LIN {X 0.053,Y -179.837,Z 893.459,A 0.000,B 0.000,C 90.000,E1 262.648} C_DIS
LIN {X -0.069,Y -179.024,Z 893.445,A 0.000,B 0.000,C 90.000,E1 260.151} C_DIS
LIN {X -0.006,Y -178.664,Z 893.440,A 0.000,B 0.000,C 90.000,E1 259.285} C_DIS
LIN {X -0.070,Y -175.715,Z 893.412,A 0.000,B 0.000,C 90.000,E1 254.212} C_DIS
LIN {X -0.053,Y -172.430,Z 893.388,A 0.000,B 0.000,C 90.000,E1 249.934} C_DIS
LIN {X -0.035,Y -171.257,Z 893.379,A 0.000,B 0.000,C 90.000,E1 248.209} C_DIS
LIN {X -0.051,Y -167.530,Z 893.355,A 0.000,B 0.000,C 90.000,E1 243.896} C_DIS
LIN {X 0.033,Y -166.925,Z 893.350,A 0.000,B 0.000,C 90.000,E1 242.999} C_DIS
LIN {X -0.046,Y -162.921,Z 893.326,A 0.000,B 0.000,C 90.000,E1 238.663} C_DIS
LIN {X -0.068,Y -161.594,Z 893.316,A 0.000,B 0.000,C 90.000,E1 236.914} C_DIS
LIN {X 0.057,Y -158.336,Z 893.296,A 0.000,B 0.000,C 90.000,E1 233.336} C_DIS
LIN {X -0.081,Y -155.638,Z 893.277,A 0.000,B 0.000,C 90.000,E1 229.828} C_DIS
LIN {X -0.027,Y -151.912,Z 893.252,A 0.000,B 0.000,C 90.000,E1 225.324} C_DIS
LIN {X -0.012,Y -150.145,Z 893.237,A 0.000,B 0.000,C 90.000,E1 222.609} C_DIS
LIN {X 0.025,Y -146.929,Z 893.211,A 0.000,B 0.000,C 90.000,E1 218.051} C_DIS
LIN {X 0.017,Y -145.517,Z 893.196,A 0.000,B 0.000,C 90.000,E1 215.311} C_DIS
LIN {X 0.011,Y -142.917,Z 893.171,A 0.000,B 0.000,C 90.000,E1 210.718} C_DIS
LIN {X 0.064,Y -141.540,Z 893.150,A 0.000,B 0.000,C 90.000,E1 207.001} C_DIS
LIN {X -0.024,Y -139.402,Z 893.114,A 0.000,B 0.000,C 90.000,E1 200.536} C_DIS
LIN {X -0.019,Y -139.118,Z 893.104,A 0.000,B 0.000,C 90.000,E1 198.671} C_DIS
LIN {X 0.012,Y -138.352,Z 893.057,A 0.000,B 0.000,C 90.000,E1 190.254} C_DIS
LIN {X 0.002,Y -139.505,Z 893.005,A 0.000,B 0.000,C 90.000,E1 180.917} C_DIS
LIN {X -0.057,Y -141.138,Z 892.974,A 0.000,B 0.000,C 90.000,E1 175.355} C_DIS
LIN {X 0.037,Y -142.518,Z 892.959,A 0.000,B 0.000,C 90.000,E1 172.534} C_DIS
LIN {X -0.018,Y -144.781,Z 892.933,A 0.000,B 0.000,C 90.000,E1 167.937} C_DIS
LIN {X -0.029,Y -147.396,Z 892.913,A 0.000,B 0.000,C 90.000,E1 164.267} C_DIS
LIN {X 0.001,Y -149.971,Z 892.892,A 0.000,B 0.000,C 90.000,E1 160.604} C_DIS
LIN {X 0.012,Y -153.292,Z 892.872,A 0.000,B 0.000,C 90.000,E1 156.975} C_DIS
LIN {X -0.001,Y -154.996,Z 892.862,A 0.000,B 0.000,C 90.000,E1 155.177} C_DIS
LIN {X 0.012,Y -158.636,Z 892.842,A 0.000,B 0.000,C 90.000,E1 151.591} C_DIS
LIN {X -0.051,Y -161.910,Z 892.827,A 0.000,B 0.000,C 90.000,E1 148.948} C_DIS
LIN {X 0.056,Y -166.101,Z 892.808,A 0.000,B 0.000,C 90.000,E1 145.388} C_DIS
LIN {X 0.054,Y -171.110,Z 892.788,A 0.000,B 0.000,C 90.000,E1 141.904} C_DIS
LIN {X -0.026,Y -175.985,Z 892.769,A 0.000,B 0.000,C 90.000,E1 138.485} C_DIS
LIN {X 0.088,Y -180.231,Z 892.755,A 0.000,B 0.000,C 90.000,E1 135.891} C_DIS
LIN {X 0.061,Y -185.646,Z 892.736,A 0.000,B 0.000,C 90.000,E1 132.528} C_DIS
LIN {X 0.115,Y -190.245,Z 892.722,A 0.000,B 0.000,C 90.000,E1 130.011} C_DIS
LIN {X -0.048,Y -193.381,Z 892.712,A 0.000,B 0.000,C 90.000,E1 128.222} C_DIS
LIN {X 0.109,Y -294.897,Z 892.712,A 0.000,B 0.000,C 90.000,E1 128.177} C_DIS
LIN {X 0.093,Y -299.925,Z 892.711,A 0.000,B 0.000,C 90.000,E1 128.016} C_DIS
LIN {X -0.060,Y -302.135,Z 892.710,A 0.000,B 0.000,C 90.000,E1 127.890} C_DIS
LIN {X 0.005,Y -305.159,Z 892.709,A 0.000,B 0.000,C 90.000,E1 127.569} C_DIS
LIN {X -0.008,Y -308.784,Z 892.706,A 0.000,B 0.000,C 90.000,E1 126.996} C_DIS
LIN {X 0.017,Y -310.226,Z 892.704,A 0.000,B 0.000,C 90.000,E1 126.664} C_DIS
LIN {X -0.023,Y -311.357,Z 892.702,A 0.000,B 0.000,C 90.000,E1 126.343} C_DIS
LIN {X 0.139,Y -321.511,Z 892.684,A 0.000,B 0.000,C 90.000,E1 123.086} C_DIS
LIN {X 0.013,Y -331.967,Z 892.668,A 0.000,B 0.000,C 90.000,E1 120.256} C_DIS
LIN {X -0.023,Y -343.778,Z 892.653,A 0.000,B 0.000,C 90.000,E1 117.462} C_DIS
LIN {X -0.023,Y -357.045,Z 892.637,A 0.000,B 0.000,C 90.000,E1 114.719} C_DIS
LIN {X -0.034,Y -370.158,Z 892.624,A 0.000,B 0.000,C 90.000,E1 112.333} C_DIS
LIN {X -0.006,Y -384.610,Z 892.611,A 0.000,B 0.000,C 90.000,E1 109.993} C_DIS
LIN {X 0.121,Y -400.503,Z 892.598,A 0.000,B 0.000,C 90.000,E1 107.692} C_DIS
LIN {X 0.017,Y -417.952,Z 892.586,A 0.000,B 0.000,C 90.000,E1 105.481} C_DIS
LIN {X 0.148,Y -437.059,Z 892.574,A 0.000,B 0.000,C 90.000,E1 103.300} C_DIS
LIN {X -0.056,Y -457.177,Z 892.563,A 0.000,B 0.000,C 90.000,E1 101.299} C_DIS
LIN {X -0.201,Y -467.395,Z 892.557,A 0.000,B 0.000,C 90.000,E1 100.366} C_DIS
LIN {X -0.258,Y -469.394,Z 892.556,A 0.000,B 0.000,C 90.000,E1 100.141} C_DIS
LIN {X 0.054,Y -471.044,Z 892.555,A 0.000,B 0.000,C 90.000,E1 99.849} C_DIS
LIN {X -0.099,Y -472.281,Z 892.553,A 0.000,B 0.000,C 90.000,E1 99.613} C_DIS
LIN {X 0.005,Y -473.801,Z 892.551,A 0.000,B 0.000,C 90.000,E1 99.095} C_DIS
LIN {X 0.191,Y -474.280,Z 892.548,A 0.000,B 0.000,C 90.000,E1 98.568} C_DIS
LIN {X -0.155,Y -473.796,Z 892.545,A 0.000,B 0.000,C 90.000,E1 98.106} C_DIS
LIN {X -0.028,Y -472.278,Z 892.542,A 0.000,B 0.000,C 90.000,E1 97.587} C_DIS
LIN {X -0.169,Y -471.051,Z 892.541,A 0.000,B 0.000,C 90.000,E1 97.352} C_DIS
LIN {X 0.203,Y -452.056,Z 892.524,A 0.000,B 0.000,C 90.000,E1 94.245} C_DIS
LIN {X 0.123,Y -443.002,Z 892.515,A 0.000,B 0.000,C 90.000,E1 92.694} C_DIS
LIN {X -0.134,Y -433.515,Z 892.506,A 0.000,B 0.000,C 90.000,E1 91.146} C_DIS
LIN {X -0.125,Y -423.861,Z 892.497,A 0.000,B 0.000,C 90.000,E1 89.542} C_DIS
LIN {X -0.091,Y -410.897,Z 892.485,A 0.000,B 0.000,C 90.000,E1 87.364} C_DIS
LIN {X 0.014,Y -399.646,Z 892.475,A 0.000,B 0.000,C 90.000,E1 85.412} C_DIS
LIN {X -0.043,Y -386.908,Z 892.462,A 0.000,B 0.000,C 90.000,E1 83.166} C_DIS
LIN {X 0.063,Y -375.774,Z 892.451,A 0.000,B 0.000,C 90.000,E1 81.141} C_DIS
LIN {X -0.003,Y -364.602,Z 892.439,A 0.000,B 0.000,C 90.000,E1 79.106} C_DIS
LIN {X -0.188,Y -354.940,Z 892.430,A 0.000,B 0.000,C 90.000,E1 77.353} C_DIS
LIN {X -0.122,Y -343.614,Z 892.418,A 0.000,B 0.000,C 90.000,E1 75.227} C_DIS
LIN {X 0.088,Y -330.953,Z 892.404,A 0.000,B 0.000,C 90.000,E1 72.725} C_DIS
LIN {X 0.056,Y -315.972,Z 892.387,A 0.000,B 0.000,C 90.000,E1 69.571} C_DIS
LIN {X 0.090,Y -305.677,Z 892.374,A 0.000,B 0.000,C 90.000,E1 67.305} C_DIS
LIN {X -0.024,Y -295.551,Z 892.361,A 0.000,B 0.000,C 90.000,E1 65.025} C_DIS
LIN {X 0.052,Y -285.342,Z 892.348,A 0.000,B 0.000,C 90.000,E1 62.666} C_DIS
LIN {X -0.037,Y -276.501,Z 892.337,A 0.000,B 0.000,C 90.000,E1 60.639} C_DIS
LIN {X -0.096,Y -262.185,Z 892.318,A 0.000,B 0.000,C 90.000,E1 57.168} C_DIS
LIN {X 0.091,Y -250.354,Z 892.300,A 0.000,B 0.000,C 90.000,E1 53.909} C_DIS
LIN {X 0.005,Y -242.092,Z 892.285,A 0.000,B 0.000,C 90.000,E1 51.376} C_DIS
LIN {X 0.022,Y -233.427,Z 892.269,A 0.000,B 0.000,C 90.000,E1 48.405} C_DIS
LIN {X -0.008,Y -223.518,Z 892.248,A 0.000,B 0.000,C 90.000,E1 44.636} C_DIS
LIN {X -0.008,Y -214.259,Z 892.227,A 0.000,B 0.000,C 90.000,E1 40.782} C_DIS
LIN {X -0.025,Y -207.358,Z 892.209,A 0.000,B 0.000,C 90.000,E1 37.649} C_DIS
LIN {X 0.019,Y -200.922,Z 892.191,A 0.000,B 0.000,C 90.000,E1 34.452} C_DIS
LIN {X 0.067,Y -195.005,Z 892.174,A 0.000,B 0.000,C 90.000,E1 31.209} C_DIS
LIN {X -0.055,Y -189.675,Z 892.155,A 0.000,B 0.000,C 90.000,E1 27.975} C_DIS
LIN {X 0.017,Y -185.015,Z 892.137,A 0.000,B 0.000,C 90.000,E1 24.643} C_DIS
LIN {X -0.060,Y -180.142,Z 892.114,A 0.000,B 0.000,C 90.000,E1 20.482} C_DIS
LIN {X -0.082,Y -176.382,Z 892.090,A 0.000,B 0.000,C 90.000,E1 16.260} C_DIS
LIN {X -0.054,Y -173.296,Z 892.062,A 0.000,B 0.000,C 90.000,E1 11.130} C_DIS
LIN {X -0.024,Y -171.478,Z 892.014,A 0.000,B 0.000,C 90.000,E1 2.522} C_DIS
LIN {X -0.017,Y -173.366,Z 891.969,A 0.000,B 0.000,C 90.000,E1 354.375} C_DIS
LIN {X -0.032,Y -175.801,Z 891.945,A 0.000,B 0.000,C 90.000,E1 350.095} C_DIS
LIN {X 0.004,Y -179.225,Z 891.921,A 0.000,B 0.000,C 90.000,E1 345.825} C_DIS
LIN {X 0.088,Y -182.848,Z 891.902,A 0.000,B 0.000,C 90.000,E1 342.417} C_DIS
LIN {X 0.032,Y -187.234,Z 891.884,A 0.000,B 0.000,C 90.000,E1 339.082} C_DIS
LIN {X -0.067,Y -192.413,Z 891.865,A 0.000,B 0.000,C 90.000,E1 335.793} C_DIS
LIN {X 0.023,Y -198.295,Z 891.847,A 0.000,B 0.000,C 90.000,E1 332.487} C_DIS
LIN {X 0.015,Y -204.536,Z 891.829,A 0.000,B 0.000,C 90.000,E1 329.253} C_DIS
LIN {X -0.085,Y -211.251,Z 891.811,A 0.000,B 0.000,C 90.000,E1 326.087} C_DIS
LIN {X -0.020,Y -218.410,Z 891.794,A 0.000,B 0.000,C 90.000,E1 322.924} C_DIS
LIN {X -0.090,Y -227.187,Z 891.775,A 0.000,B 0.000,C 90.000,E1 319.461} C_DIS
LIN {X 0.110,Y -235.870,Z 891.758,A 0.000,B 0.000,C 90.000,E1 316.377} C_DIS
LIN {X 0.002,Y -246.823,Z 891.739,A 0.000,B 0.000,C 90.000,E1 313.056} C_DIS
LIN {X -0.130,Y -257.648,Z 891.723,A 0.000,B 0.000,C 90.000,E1 310.172} C_DIS
LIN {X -0.036,Y -271.020,Z 891.705,A 0.000,B 0.000,C 90.000,E1 306.950} C_DIS
LIN {X -0.048,Y -285.676,Z 891.688,A 0.000,B 0.000,C 90.000,E1 303.833} C_DIS
LIN {X -0.028,Y -301.730,Z 891.671,A 0.000,B 0.000,C 90.000,E1 300.797} C_DIS
LIN {X 0.097,Y -317.463,Z 891.656,A 0.000,B 0.000,C 90.000,E1 298.153} C_DIS
LIN {X 0.123,Y -330.363,Z 891.646,A 0.000,B 0.000,C 90.000,E1 296.232} C_DIS
LIN {X -0.050,Y -344.471,Z 891.635,A 0.000,B 0.000,C 90.000,E1 294.387} C_DIS
LIN {X -0.012,Y -364.459,Z 891.622,A 0.000,B 0.000,C 90.000,E1 291.950} C_DIS
LIN {X 0.175,Y -382.277,Z 891.611,A 0.000,B 0.000,C 90.000,E1 289.939} C_DIS
LIN {X -0.038,Y -400.275,Z 891.600,A 0.000,B 0.000,C 90.000,E1 288.055} C_DIS
LIN {X 0.210,Y -413.101,Z 891.593,A 0.000,B 0.000,C 90.000,E1 286.677} C_DIS
LIN {X 0.066,Y -425.496,Z 891.585,A 0.000,B 0.000,C 90.000,E1 285.371} C_DIS
LIN {X 0.015,Y -435.194,Z 891.579,A 0.000,B 0.000,C 90.000,E1 284.300} C_DIS
LIN {X -0.043,Y -444.486,Z 891.574,A 0.000,B 0.000,C 90.000,E1 283.244} C_DIS
LIN {X -0.182,Y -455.344,Z 891.566,A 0.000,B 0.000,C 90.000,E1 281.951} C_DIS
LIN {X -0.001,Y -463.374,Z 891.561,A 0.000,B 0.000,C 90.000,E1 280.894} C_DIS
LIN {X 0.045,Y -472.588,Z 891.553,A 0.000,B 0.000,C 90.000,E1 279.613} C_DIS
LIN {X 0.008,Y -477.641,Z 891.549,A 0.000,B 0.000,C 90.000,E1 278.859} C_DIS
LIN {X 0.021,Y -481.992,Z 891.545,A 0.000,B 0.000,C 90.000,E1 278.106} C_DIS
LIN {X 0.066,Y -485.666,Z 891.541,A 0.000,B 0.000,C 90.000,E1 277.352} C_DIS
LIN {X -0.228,Y -487.704,Z 891.538,A 0.000,B 0.000,C 90.000,E1 276.891} C_DIS
LIN {X -0.032,Y -489.390,Z 891.535,A 0.000,B 0.000,C 90.000,E1 276.372} C_DIS
LIN {X 0.178,Y -490.721,Z 891.533,A 0.000,B 0.000,C 90.000,E1 275.853} C_DIS
LIN {X -0.092,Y -491.768,Z 891.530,A 0.000,B 0.000,C 90.000,E1 275.391} C_DIS
LIN {X 0.092,Y -492.352,Z 891.527,A 0.000,B 0.000,C 90.000,E1 274.878} C_DIS
LIN {X -0.166,Y -492.530,Z 891.524,A 0.000,B 0.000,C 90.000,E1 274.416} C_DIS
LIN {X 0.067,Y -492.285,Z 891.522,A 0.000,B 0.000,C 90.000,E1 273.898} C_DIS
LIN {X -0.222,Y -491.625,Z 891.519,A 0.000,B 0.000,C 90.000,E1 273.440} C_DIS
LIN {X 0.008,Y -490.491,Z 891.516,A 0.000,B 0.000,C 90.000,E1 272.922} C_DIS
LIN {X 0.208,Y -488.882,Z 891.513,A 0.000,B 0.000,C 90.000,E1 272.407} C_DIS
LIN {X -0.084,Y -486.720,Z 891.511,A 0.000,B 0.000,C 90.000,E1 271.949} C_DIS
LIN {X 0.117,Y -483.965,Z 891.508,A 0.000,B 0.000,C 90.000,E1 271.432} C_DIS
LIN {X -0.200,Y -480.429,Z 891.505,A 0.000,B 0.000,C 90.000,E1 270.974} C_DIS
LIN {X -0.051,Y -476.057,Z 891.503,A 0.000,B 0.000,C 90.000,E1 270.458} C_DIS
LIN {X 0.074,Y -470.645,Z 891.500,A 0.000,B 0.000,C 90.000,E1 269.943} C_DIS
LIN {X 0.080,Y -464.678,Z 891.497,A 0.000,B 0.000,C 90.000,E1 269.484} C_DIS
LIN {X 0.125,Y -458.426,Z 891.495,A 0.000,B 0.000,C 90.000,E1 269.083} C_DIS
LIN {X 0.115,Y -451.796,Z 891.493,A 0.000,B 0.000,C 90.000,E1 268.740} C_DIS
LIN {X 0.013,Y -444.622,Z 891.491,A 0.000,B 0.000,C 90.000,E1 268.453} C_DIS
LIN {X -0.105,Y -437.329,Z 891.490,A 0.000,B 0.000,C 90.000,E1 268.224} C_DIS
LIN {X 0.158,Y -429.411,Z 891.489,A 0.000,B 0.000,C 90.000,E1 267.993} C_DIS
LIN {X -0.079,Y -421.239,Z 891.488,A 0.000,B 0.000,C 90.000,E1 267.879} C_DIS
LIN {X 0.170,Y -413.473,Z 891.488,A 0.000,B 0.000,C 90.000,E1 267.764} C_DIS
LIN {X -0.022,Y -408.253,Z 891.488,A 0.000,B 0.000,C 90.000,E1 267.764} C_DIS
LIN {X -0.032,Y -181.086,Z 891.488,A 0.000,B 0.000,C 90.000,E1 267.764} C_DIS
LIN {X -0.011,Y -180.893,Z 891.473,A 0.000,B 0.000,C 90.000,E1 265.179} C_DIS
LIN {X 0.066,Y -179.516,Z 891.454,A 0.000,B 0.000,C 90.000,E1 261.781} C_DIS
LIN {X 0.051,Y -179.020,Z 891.445,A 0.000,B 0.000,C 90.000,E1 260.095} C_DIS
LIN {X -0.030,Y -178.652,Z 891.440,A 0.000,B 0.000,C 90.000,E1 259.275} C_DIS
LIN {X 0.043,Y -175.703,Z 891.412,A 0.000,B 0.000,C 90.000,E1 254.157} C_DIS
LIN {X 0.053,Y -172.419,Z 891.388,A 0.000,B 0.000,C 90.000,E1 249.880} C_DIS
LIN {X 0.070,Y -171.239,Z 891.379,A 0.000,B 0.000,C 90.000,E1 248.156} C_DIS
LIN {X 0.045,Y -167.517,Z 891.355,A 0.000,B 0.000,C 90.000,E1 243.845} C_DIS
LIN {X -0.023,Y -166.911,Z 891.350,A 0.000,B 0.000,C 90.000,E1 242.999} C_DIS
LIN {X 0.029,Y -162.220,Z 891.321,A 0.000,B 0.000,C 90.000,E1 237.740} C_DIS
LIN {X -0.051,Y -160.800,Z 891.311,A 0.000,B 0.000,C 90.000,E1 236.008} C_DIS
LIN {X -0.071,Y -157.588,Z 891.291,A 0.000,B 0.000,C 90.000,E1 232.477} C_DIS
LIN {X -0.014,Y -155.621,Z 891.277,A 0.000,B 0.000,C 90.000,E1 229.784} C_DIS
LIN {X -0.079,Y -151.898,Z 891.252,A 0.000,B 0.000,C 90.000,E1 225.324} C_DIS
LIN {X -0.063,Y -150.128,Z 891.237,A 0.000,B 0.000,C 90.000,E1 222.609} C_DIS
LIN {X 0.065,Y -146.917,Z 891.211,A 0.000,B 0.000,C 90.000,E1 218.016} C_DIS
LIN {X -0.034,Y -145.506,Z 891.196,A 0.000,B 0.000,C 90.000,E1 215.311} C_DIS
LIN {X -0.039,Y -142.909,Z 891.171,A 0.000,B 0.000,C 90.000,E1 210.718} C_DIS
LIN {X 0.014,Y -141.530,Z 891.150,A 0.000,B 0.000,C 90.000,E1 207.001} C_DIS
LIN {X 0.057,Y -139.399,Z 891.114,A 0.000,B 0.000,C 90.000,E1 200.482} C_DIS
LIN {X -0.024,Y -139.112,Z 891.104,A 0.000,B 0.000,C 90.000,E1 198.652} C_DIS
LIN {X -0.037,Y -138.353,Z 891.057,A 0.000,B 0.000,C 90.000,E1 190.254} C_DIS
LIN {X -0.047,Y -139.507,Z 891.005,A 0.000,B 0.000,C 90.000,E1 180.917} C_DIS
LIN {X 0.034,Y -141.147,Z 890.974,A 0.000,B 0.000,C 90.000,E1 175.298} C_DIS
LIN {X -0.013,Y -142.527,Z 890.958,A 0.000,B 0.000,C 90.000,E1 172.534} C_DIS
LIN {X -0.067,Y -144.792,Z 890.933,A 0.000,B 0.000,C 90.000,E1 167.937} C_DIS
LIN {X 0.062,Y -147.410,Z 890.912,A 0.000,B 0.000,C 90.000,E1 164.212} C_DIS
LIN {X -0.050,Y -149.987,Z 890.892,A 0.000,B 0.000,C 90.000,E1 160.604} C_DIS
LIN {X -0.041,Y -153.312,Z 890.872,A 0.000,B 0.000,C 90.000,E1 156.975} C_DIS
LIN {X 0.012,Y -155.013,Z 890.862,A 0.000,B 0.000,C 90.000,E1 155.153} C_DIS
LIN {X 0.034,Y -158.658,Z 890.842,A 0.000,B 0.000,C 90.000,E1 151.563} C_DIS
LIN {X -0.022,Y -161.935,Z 890.827,A 0.000,B 0.000,C 90.000,E1 148.918} C_DIS
LIN {X 0.002,Y -166.125,Z 890.808,A 0.000,B 0.000,C 90.000,E1 145.388} C_DIS
LIN {X -0.001,Y -171.137,Z 890.788,A 0.000,B 0.000,C 90.000,E1 141.904} C_DIS
LIN {X 0.034,Y -176.014,Z 890.769,A 0.000,B 0.000,C 90.000,E1 138.447} C_DIS
LIN {X 0.030,Y -180.265,Z 890.755,A 0.000,B 0.000,C 90.000,E1 135.891} C_DIS
LIN {X 0.002,Y -185.678,Z 890.736,A 0.000,B 0.000,C 90.000,E1 132.528} C_DIS
LIN {X 0.055,Y -190.280,Z 890.722,A 0.000,B 0.000,C 90.000,E1 130.011} C_DIS
LIN {X -0.018,Y -193.366,Z 890.712,A 0.000,B 0.000,C 90.000,E1 128.222} C_DIS
LIN {X -0.063,Y -295.099,Z 890.712,A 0.000,B 0.000,C 90.000,E1 128.222} C_DIS
LIN {X -0.033,Y -297.042,Z 890.712,A 0.000,B 0.000,C 90.000,E1 128.177} C_DIS
LIN {X 0.032,Y -302.451,Z 890.710,A 0.000,B 0.000,C 90.000,E1 127.855} C_DIS
LIN {X 0.152,Y -305.353,Z 890.709,A 0.000,B 0.000,C 90.000,E1 127.523} C_DIS
LIN {X 0.099,Y -307.382,Z 890.707,A 0.000,B 0.000,C 90.000,E1 127.237} C_DIS
LIN {X 0.044,Y -308.968,Z 890.705,A 0.000,B 0.000,C 90.000,E1 126.950} C_DIS
LIN {X -0.172,Y -310.352,Z 890.703,A 0.000,B 0.000,C 90.000,E1 126.664} C_DIS
LIN {X -0.097,Y -315.325,Z 890.694,A 0.000,B 0.000,C 90.000,E1 125.025} C_DIS
LIN {X 0.031,Y -326.095,Z 890.677,A 0.000,B 0.000,C 90.000,E1 121.799} C_DIS
LIN {X 0.156,Y -337.155,Z 890.661,A 0.000,B 0.000,C 90.000,E1 118.949} C_DIS
LIN {X -0.194,Y -349.619,Z 890.646,A 0.000,B 0.000,C 90.000,E1 116.232} C_DIS
LIN {X -0.191,Y -363.588,Z 890.630,A 0.000,B 0.000,C 90.000,E1 113.515} C_DIS
LIN {X 0.156,Y -377.375,Z 890.617,A 0.000,B 0.000,C 90.000,E1 111.099} C_DIS
LIN {X 0.239,Y -392.553,Z 890.604,A 0.000,B 0.000,C 90.000,E1 108.779} C_DIS
LIN {X 0.064,Y -409.228,Z 890.592,A 0.000,B 0.000,C 90.000,E1 106.551} C_DIS
LIN {X 0.061,Y -427.524,Z 890.580,A 0.000,B 0.000,C 90.000,E1 104.356} C_DIS
LIN {X 0.106,Y -447.284,Z 890.568,A 0.000,B 0.000,C 90.000,E1 102.243} C_DIS
LIN {X 0.057,Y -467.610,Z 890.557,A 0.000,B 0.000,C 90.000,E1 100.310} C_DIS
LIN {X 0.085,Y -469.556,Z 890.556,A 0.000,B 0.000,C 90.000,E1 100.074} C_DIS
LIN {X -0.147,Y -471.164,Z 890.555,A 0.000,B 0.000,C 90.000,E1 99.849} C_DIS
LIN {X 0.166,Y -472.371,Z 890.553,A 0.000,B 0.000,C 90.000,E1 99.557} C_DIS
LIN {X -0.195,Y -473.842,Z 890.550,A 0.000,B 0.000,C 90.000,E1 99.095} C_DIS
LIN {X -0.009,Y -474.279,Z 890.548,A 0.000,B 0.000,C 90.000,E1 98.568} C_DIS
LIN {X 0.114,Y -473.754,Z 890.545,A 0.000,B 0.000,C 90.000,E1 98.049} C_DIS
LIN {X -0.228,Y -472.188,Z 890.542,A 0.000,B 0.000,C 90.000,E1 97.587} C_DIS
LIN {X 0.098,Y -470.931,Z 890.541,A 0.000,B 0.000,C 90.000,E1 97.296} C_DIS
LIN {X 0.007,Y -451.932,Z 890.524,A 0.000,B 0.000,C 90.000,E1 94.245} C_DIS
LIN {X -0.069,Y -442.904,Z 890.515,A 0.000,B 0.000,C 90.000,E1 92.694} C_DIS
LIN {X 0.109,Y -433.410,Z 890.506,A 0.000,B 0.000,C 90.000,E1 91.088} C_DIS
LIN {X 0.110,Y -423.767,Z 890.497,A 0.000,B 0.000,C 90.000,E1 89.484} C_DIS
LIN {X 0.134,Y -410.786,Z 890.485,A 0.000,B 0.000,C 90.000,E1 87.306} C_DIS
LIN {X -0.167,Y -399.509,Z 890.474,A 0.000,B 0.000,C 90.000,E1 85.412} C_DIS
LIN {X 0.161,Y -386.770,Z 890.462,A 0.000,B 0.000,C 90.000,E1 83.109} C_DIS
LIN {X -0.115,Y -375.606,Z 890.451,A 0.000,B 0.000,C 90.000,E1 81.141} C_DIS
LIN {X -0.179,Y -364.459,Z 890.439,A 0.000,B 0.000,C 90.000,E1 79.106} C_DIS
LIN {X -0.015,Y -354.836,Z 890.429,A 0.000,B 0.000,C 90.000,E1 77.297} C_DIS
LIN {X 0.047,Y -341.926,Z 890.416,A 0.000,B 0.000,C 90.000,E1 74.866} C_DIS
LIN {X 0.080,Y -327.834,Z 890.400,A 0.000,B 0.000,C 90.000,E1 72.072} C_DIS
LIN {X -0.104,Y -315.944,Z 890.386,A 0.000,B 0.000,C 90.000,E1 69.571} C_DIS
LIN {X 0.053,Y -305.656,Z 890.374,A 0.000,B 0.000,C 90.000,E1 67.283} C_DIS
LIN {X 0.093,Y -296.991,Z 890.363,A 0.000,B 0.000,C 90.000,E1 65.305} C_DIS
LIN {X -0.075,Y -286.802,Z 890.350,A 0.000,B 0.000,C 90.000,E1 62.999} C_DIS
LIN {X 0.107,Y -278.012,Z 890.339,A 0.000,B 0.000,C 90.000,E1 60.923} C_DIS
LIN {X 0.163,Y -265.037,Z 890.321,A 0.000,B 0.000,C 90.000,E1 57.788} C_DIS
LIN {X 0.064,Y -253.040,Z 890.303,A 0.000,B 0.000,C 90.000,E1 54.609} C_DIS
LIN {X 0.082,Y -244.527,Z 890.289,A 0.000,B 0.000,C 90.000,E1 52.065} C_DIS
LIN {X -0.034,Y -235.730,Z 890.273,A 0.000,B 0.000,C 90.000,E1 49.138} C_DIS
LIN {X -0.023,Y -227.597,Z 890.256,A 0.000,B 0.000,C 90.000,E1 46.134} C_DIS
LIN {X -0.067,Y -219.928,Z 890.239,A 0.000,B 0.000,C 90.000,E1 43.095} C_DIS
LIN {X 0.039,Y -212.723,Z 890.222,A 0.000,B 0.000,C 90.000,E1 39.967} C_DIS
LIN {X 0.020,Y -205.936,Z 890.205,A 0.000,B 0.000,C 90.000,E1 36.824} C_DIS
LIN {X 0.032,Y -199.614,Z 890.187,A 0.000,B 0.000,C 90.000,E1 33.627} C_DIS
LIN {X 0.046,Y -193.846,Z 890.169,A 0.000,B 0.000,C 90.000,E1 30.384} C_DIS
LIN {X -0.033,Y -188.681,Z 890.151,A 0.000,B 0.000,C 90.000,E1 27.129} C_DIS
LIN {X -0.068,Y -184.201,Z 890.132,A 0.000,B 0.000,C 90.000,E1 23.823} C_DIS
LIN {X -0.067,Y -179.522,Z 890.109,A 0.000,B 0.000,C 90.000,E1 19.631} C_DIS
LIN {X 0.009,Y -176.010,Z 890.085,A 0.000,B 0.000,C 90.000,E1 15.371} C_DIS
LIN {X -0.013,Y -173.208,Z 890.057,A 0.000,B 0.000,C 90.000,E1 10.254} C_DIS
LIN {X 0.000,Y -174.030,Z 889.964,A 0.000,B 0.000,C 90.000,E1 353.514} C_DIS
LIN {X 0.058,Y -176.706,Z 889.940,A 0.000,B 0.000,C 90.000,E1 349.218} C_DIS
LIN {X -0.010,Y -180.366,Z 889.917,A 0.000,B 0.000,C 90.000,E1 344.991} C_DIS
LIN {X -0.071,Y -184.195,Z 889.898,A 0.000,B 0.000,C 90.000,E1 341.638} C_DIS
LIN {X -0.034,Y -188.838,Z 889.879,A 0.000,B 0.000,C 90.000,E1 338.284} C_DIS
LIN {X -0.020,Y -194.196,Z 889.861,A 0.000,B 0.000,C 90.000,E1 334.973} C_DIS
LIN {X 0.031,Y -200.175,Z 889.843,A 0.000,B 0.000,C 90.000,E1 331.691} C_DIS
LIN {X 0.074,Y -206.529,Z 889.825,A 0.000,B 0.000,C 90.000,E1 328.456} C_DIS
LIN {X -0.037,Y -213.290,Z 889.807,A 0.000,B 0.000,C 90.000,E1 325.308} C_DIS
LIN {X -0.092,Y -220.591,Z 889.790,A 0.000,B 0.000,C 90.000,E1 322.190} C_DIS
LIN {X 0.054,Y -229.528,Z 889.771,A 0.000,B 0.000,C 90.000,E1 318.690} C_DIS
LIN {X -0.016,Y -238.470,Z 889.754,A 0.000,B 0.000,C 90.000,E1 315.688} C_DIS
LIN {X 0.137,Y -248.358,Z 889.737,A 0.000,B 0.000,C 90.000,E1 312.690} C_DIS
LIN {X 0.055,Y -259.290,Z 889.721,A 0.000,B 0.000,C 90.000,E1 309.806} C_DIS
LIN {X -0.016,Y -272.727,Z 889.703,A 0.000,B 0.000,C 90.000,E1 306.629} C_DIS
LIN {X 0.093,Y -287.458,Z 889.686,A 0.000,B 0.000,C 90.000,E1 303.499} C_DIS
LIN {X 0.172,Y -303.595,Z 889.669,A 0.000,B 0.000,C 90.000,E1 300.463} C_DIS
LIN {X -0.078,Y -319.430,Z 889.655,A 0.000,B 0.000,C 90.000,E1 297.897} C_DIS
LIN {X -0.019,Y -332.455,Z 889.644,A 0.000,B 0.000,C 90.000,E1 295.976} C_DIS
LIN {X 0.155,Y -346.647,Z 889.634,A 0.000,B 0.000,C 90.000,E1 294.079} C_DIS
LIN {X 0.126,Y -366.661,Z 889.620,A 0.000,B 0.000,C 90.000,E1 291.663} C_DIS
LIN {X -0.042,Y -384.552,Z 889.609,A 0.000,B 0.000,C 90.000,E1 289.704} C_DIS
LIN {X -0.184,Y -402.574,Z 889.599,A 0.000,B 0.000,C 90.000,E1 287.819} C_DIS
LIN {X 0.067,Y -415.363,Z 889.591,A 0.000,B 0.000,C 90.000,E1 286.441} C_DIS
LIN {X 0.032,Y -425.386,Z 889.585,A 0.000,B 0.000,C 90.000,E1 285.371} C_DIS
LIN {X -0.017,Y -435.106,Z 889.579,A 0.000,B 0.000,C 90.000,E1 284.300} C_DIS
LIN {X -0.069,Y -444.388,Z 889.574,A 0.000,B 0.000,C 90.000,E1 283.244} C_DIS
LIN {X -0.211,Y -455.288,Z 889.566,A 0.000,B 0.000,C 90.000,E1 281.951} C_DIS
LIN {X -0.031,Y -463.350,Z 889.560,A 0.000,B 0.000,C 90.000,E1 280.894} C_DIS
LIN {X 0.014,Y -472.582,Z 889.553,A 0.000,B 0.000,C 90.000,E1 279.613} C_DIS
LIN {X -0.023,Y -477.600,Z 889.549,A 0.000,B 0.000,C 90.000,E1 278.859} C_DIS
LIN {X -0.011,Y -482.004,Z 889.545,A 0.000,B 0.000,C 90.000,E1 278.106} C_DIS
LIN {X 0.034,Y -485.684,Z 889.541,A 0.000,B 0.000,C 90.000,E1 277.352} C_DIS
LIN {X 0.224,Y -487.733,Z 889.538,A 0.000,B 0.000,C 90.000,E1 276.834} C_DIS
LIN {X -0.058,Y -489.444,Z 889.535,A 0.000,B 0.000,C 90.000,E1 276.372} C_DIS
LIN {X 0.152,Y -490.780,Z 889.533,A 0.000,B 0.000,C 90.000,E1 275.853} C_DIS
LIN {X -0.118,Y -491.804,Z 889.530,A 0.000,B 0.000,C 90.000,E1 275.391} C_DIS
LIN {X 0.065,Y -492.422,Z 889.527,A 0.000,B 0.000,C 90.000,E1 274.878} C_DIS
LIN {X -0.192,Y -492.605,Z 889.524,A 0.000,B 0.000,C 90.000,E1 274.416} C_DIS
LIN {X 0.042,Y -492.363,Z 889.522,A 0.000,B 0.000,C 90.000,E1 273.898} C_DIS
LIN {X -0.246,Y -491.697,Z 889.519,A 0.000,B 0.000,C 90.000,E1 273.440} C_DIS
LIN {X -0.016,Y -490.594,Z 889.516,A 0.000,B 0.000,C 90.000,E1 272.922} C_DIS
LIN {X 0.184,Y -489.036,Z 889.513,A 0.000,B 0.000,C 90.000,E1 272.407} C_DIS
LIN {X -0.107,Y -486.864,Z 889.511,A 0.000,B 0.000,C 90.000,E1 271.949} C_DIS
LIN {X 0.089,Y -484.123,Z 889.508,A 0.000,B 0.000,C 90.000,E1 271.432} C_DIS
LIN {X -0.227,Y -480.638,Z 889.505,A 0.000,B 0.000,C 90.000,E1 270.974} C_DIS
LIN {X -0.076,Y -476.306,Z 889.503,A 0.000,B 0.000,C 90.000,E1 270.458} C_DIS
LIN {X 0.050,Y -470.997,Z 889.500,A 0.000,B 0.000,C 90.000,E1 269.943} C_DIS
LIN {X -0.008,Y -465.006,Z 889.497,A 0.000,B 0.000,C 90.000,E1 269.484} C_DIS
LIN {X -0.047,Y -458.617,Z 889.495,A 0.000,B 0.000,C 90.000,E1 269.083} C_DIS
LIN {X -0.055,Y -452.015,Z 889.493,A 0.000,B 0.000,C 90.000,E1 268.740} C_DIS
LIN {X -0.139,Y -444.988,Z 889.491,A 0.000,B 0.000,C 90.000,E1 268.453} C_DIS
LIN {X 0.162,Y -437.411,Z 889.490,A 0.000,B 0.000,C 90.000,E1 268.165} C_DIS
LIN {X 0.027,Y -429.904,Z 889.489,A 0.000,B 0.000,C 90.000,E1 267.993} C_DIS
LIN {X 0.209,Y -421.567,Z 889.488,A 0.000,B 0.000,C 90.000,E1 267.822} C_DIS
LIN {X 0.050,Y -414.301,Z 889.488,A 0.000,B 0.000,C 90.000,E1 267.764} C_DIS
LIN {X -0.139,Y -409.765,Z 889.487,A 0.000,B 0.000,C 90.000,E1 267.764} C_DIS
LIN {X -0.085,Y -181.084,Z 889.487,A 0.000,B 0.000,C 90.000,E1 267.764} C_DIS
LIN {X -0.071,Y -180.890,Z 889.473,A 0.000,B 0.000,C 90.000,E1 265.179} C_DIS
LIN {X -0.009,Y -179.015,Z 889.445,A 0.000,B 0.000,C 90.000,E1 260.095} C_DIS
LIN {X 0.086,Y -178.638,Z 889.440,A 0.000,B 0.000,C 90.000,E1 259.218} C_DIS
LIN {X -0.016,Y -175.690,Z 889.412,A 0.000,B 0.000,C 90.000,E1 254.157} C_DIS
LIN {X -0.005,Y -172.406,Z 889.388,A 0.000,B 0.000,C 90.000,E1 249.880} C_DIS
LIN {X 0.011,Y -171.219,Z 889.379,A 0.000,B 0.000,C 90.000,E1 248.156} C_DIS
LIN {X -0.012,Y -167.502,Z 889.355,A 0.000,B 0.000,C 90.000,E1 243.845} C_DIS
LIN {X -0.080,Y -166.898,Z 889.350,A 0.000,B 0.000,C 90.000,E1 242.999} C_DIS
LIN {X -0.027,Y -162.205,Z 889.321,A 0.000,B 0.000,C 90.000,E1 237.740} C_DIS
LIN {X 0.026,Y -160.780,Z 889.311,A 0.000,B 0.000,C 90.000,E1 235.960} C_DIS
LIN {X -0.002,Y -157.572,Z 889.291,A 0.000,B 0.000,C 90.000,E1 232.431} C_DIS
LIN {X 0.032,Y -155.604,Z 889.276,A 0.000,B 0.000,C 90.000,E1 229.747} C_DIS
LIN {X 0.082,Y -151.884,Z 889.252,A 0.000,B 0.000,C 90.000,E1 225.243} C_DIS
LIN {X 0.096,Y -150.111,Z 889.236,A 0.000,B 0.000,C 90.000,E1 222.528} C_DIS
LIN {X 0.012,Y -146.905,Z 889.211,A 0.000,B 0.000,C 90.000,E1 218.016} C_DIS
LIN {X -0.086,Y -145.493,Z 889.196,A 0.000,B 0.000,C 90.000,E1 215.311} C_DIS
LIN {X 0.032,Y -142.899,Z 889.170,A 0.000,B 0.000,C 90.000,E1 210.669} C_DIS
LIN {X -0.037,Y -141.520,Z 889.150,A 0.000,B 0.000,C 90.000,E1 207.001} C_DIS
LIN {X 0.006,Y -139.394,Z 889.114,A 0.000,B 0.000,C 90.000,E1 200.482} C_DIS
LIN {X 0.057,Y -139.105,Z 889.103,A 0.000,B 0.000,C 90.000,E1 198.598} C_DIS
LIN {X 0.049,Y -138.353,Z 889.057,A 0.000,B 0.000,C 90.000,E1 190.197} C_DIS
LIN {X 0.042,Y -139.511,Z 889.005,A 0.000,B 0.000,C 90.000,E1 180.859} C_DIS
LIN {X -0.018,Y -141.155,Z 888.974,A 0.000,B 0.000,C 90.000,E1 175.298} C_DIS
LIN {X -0.046,Y -142.536,Z 888.958,A 0.000,B 0.000,C 90.000,E1 172.527} C_DIS
LIN {X 0.022,Y -144.805,Z 888.933,A 0.000,B 0.000,C 90.000,E1 167.881} C_DIS
LIN {X 0.009,Y -147.425,Z 888.912,A 0.000,B 0.000,C 90.000,E1 164.212} C_DIS
LIN {X 0.037,Y -150.002,Z 888.892,A 0.000,B 0.000,C 90.000,E1 160.550} C_DIS
LIN {X 0.045,Y -153.333,Z 888.872,A 0.000,B 0.000,C 90.000,E1 156.922} C_DIS
LIN {X 0.027,Y -155.868,Z 888.857,A 0.000,B 0.000,C 90.000,E1 154.229} C_DIS
LIN {X -0.006,Y -159.721,Z 888.837,A 0.000,B 0.000,C 90.000,E1 150.667} C_DIS
LIN {X 0.060,Y -161.960,Z 888.827,A 0.000,B 0.000,C 90.000,E1 148.869} C_DIS
LIN {X -0.056,Y -166.151,Z 888.808,A 0.000,B 0.000,C 90.000,E1 145.388} C_DIS
LIN {X -0.060,Y -171.164,Z 888.788,A 0.000,B 0.000,C 90.000,E1 141.904} C_DIS
LIN {X -0.025,Y -176.044,Z 888.769,A 0.000,B 0.000,C 90.000,E1 138.447} C_DIS
LIN {X -0.030,Y -180.298,Z 888.755,A 0.000,B 0.000,C 90.000,E1 135.891} C_DIS
LIN {X -0.058,Y -185.710,Z 888.736,A 0.000,B 0.000,C 90.000,E1 132.528} C_DIS
LIN {X -0.007,Y -190.317,Z 888.722,A 0.000,B 0.000,C 90.000,E1 130.011} C_DIS
LIN {X -0.062,Y -193.328,Z 888.712,A 0.000,B 0.000,C 90.000,E1 128.257} C_DIS
LIN {X 0.035,Y -294.595,Z 888.712,A 0.000,B 0.000,C 90.000,E1 128.222} C_DIS
LIN {X -0.016,Y -295.510,Z 888.712,A 0.000,B 0.000,C 90.000,E1 128.222} C_DIS
LIN {X 0.165,Y -300.063,Z 888.711,A 0.000,B 0.000,C 90.000,E1 128.016} C_DIS
LIN {X -0.075,Y -302.390,Z 888.710,A 0.000,B 0.000,C 90.000,E1 127.890} C_DIS
LIN {X 0.054,Y -305.547,Z 888.708,A 0.000,B 0.000,C 90.000,E1 127.523} C_DIS
LIN {X -0.022,Y -307.540,Z 888.707,A 0.000,B 0.000,C 90.000,E1 127.237} C_DIS
LIN {X -0.100,Y -309.100,Z 888.705,A 0.000,B 0.000,C 90.000,E1 126.950} C_DIS
LIN {X 0.118,Y -310.442,Z 888.703,A 0.000,B 0.000,C 90.000,E1 126.583} C_DIS
LIN {X -0.110,Y -322.771,Z 888.682,A 0.000,B 0.000,C 90.000,E1 122.752} C_DIS
LIN {X 0.080,Y -333.401,Z 888.666,A 0.000,B 0.000,C 90.000,E1 119.873} C_DIS
LIN {X 0.096,Y -345.395,Z 888.651,A 0.000,B 0.000,C 90.000,E1 117.078} C_DIS
LIN {X 0.143,Y -358.865,Z 888.635,A 0.000,B 0.000,C 90.000,E1 114.335} C_DIS
LIN {X 0.039,Y -372.171,Z 888.622,A 0.000,B 0.000,C 90.000,E1 111.972} C_DIS
LIN {X 0.124,Y -386.829,Z 888.609,A 0.000,B 0.000,C 90.000,E1 109.631} C_DIS
LIN {X -0.192,Y -402.946,Z 888.596,A 0.000,B 0.000,C 90.000,E1 107.402} C_DIS
LIN {X 0.166,Y -420.637,Z 888.584,A 0.000,B 0.000,C 90.000,E1 105.134} C_DIS
LIN {X -0.023,Y -439.973,Z 888.572,A 0.000,B 0.000,C 90.000,E1 103.008} C_DIS
LIN {X -0.029,Y -460.175,Z 888.561,A 0.000,B 0.000,C 90.000,E1 101.007} C_DIS
LIN {X -0.105,Y -467.774,Z 888.557,A 0.000,B 0.000,C 90.000,E1 100.310} C_DIS
LIN {X -0.076,Y -469.679,Z 888.556,A 0.000,B 0.000,C 90.000,E1 100.074} C_DIS
LIN {X 0.156,Y -471.258,Z 888.555,A 0.000,B 0.000,C 90.000,E1 99.792} C_DIS
LIN {X 0.005,Y -472.441,Z 888.553,A 0.000,B 0.000,C 90.000,E1 99.557} C_DIS
LIN {X 0.186,Y -473.876,Z 888.550,A 0.000,B 0.000,C 90.000,E1 99.029} C_DIS
LIN {X -0.169,Y -474.281,Z 888.547,A 0.000,B 0.000,C 90.000,E1 98.568} C_DIS
LIN {X -0.047,Y -473.724,Z 888.545,A 0.000,B 0.000,C 90.000,E1 98.049} C_DIS
LIN {X 0.080,Y -472.121,Z 888.542,A 0.000,B 0.000,C 90.000,E1 97.530} C_DIS
LIN {X -0.060,Y -470.840,Z 888.540,A 0.000,B 0.000,C 90.000,E1 97.296} C_DIS
LIN {X 0.088,Y -453.345,Z 888.525,A 0.000,B 0.000,C 90.000,E1 94.473} C_DIS
LIN {X 0.031,Y -444.348,Z 888.516,A 0.000,B 0.000,C 90.000,E1 92.922} C_DIS
LIN {X -0.203,Y -434.931,Z 888.508,A 0.000,B 0.000,C 90.000,E1 91.375} C_DIS
LIN {X -0.170,Y -425.329,Z 888.499,A 0.000,B 0.000,C 90.000,E1 89.771} C_DIS
LIN {X -0.194,Y -413.934,Z 888.488,A 0.000,B 0.000,C 90.000,E1 87.879} C_DIS
LIN {X -0.016,Y -402.617,Z 888.477,A 0.000,B 0.000,C 90.000,E1 85.927} C_DIS
LIN {X -0.050,Y -391.390,Z 888.466,A 0.000,B 0.000,C 90.000,E1 83.970} C_DIS
LIN {X 0.111,Y -380.278,Z 888.455,A 0.000,B 0.000,C 90.000,E1 81.951} C_DIS
LIN {X 0.071,Y -369.123,Z 888.444,A 0.000,B 0.000,C 90.000,E1 79.926} C_DIS
LIN {X -0.070,Y -357.989,Z 888.433,A 0.000,B 0.000,C 90.000,E1 77.881} C_DIS
LIN {X 0.056,Y -346.671,Z 888.421,A 0.000,B 0.000,C 90.000,E1 75.755} C_DIS
LIN {X -0.072,Y -333.997,Z 888.407,A 0.000,B 0.000,C 90.000,E1 73.323} C_DIS
LIN {X -0.056,Y -320.354,Z 888.392,A 0.000,B 0.000,C 90.000,E1 70.496} C_DIS
LIN {X 0.071,Y -310.056,Z 888.379,A 0.000,B 0.000,C 90.000,E1 68.230} C_DIS
LIN {X 0.090,Y -298.458,Z 888.365,A 0.000,B 0.000,C 90.000,E1 65.613} C_DIS
LIN {X -0.040,Y -288.278,Z 888.352,A 0.000,B 0.000,C 90.000,E1 63.307} C_DIS
LIN {X 0.041,Y -279.538,Z 888.340,A 0.000,B 0.000,C 90.000,E1 61.257} C_DIS
LIN {X -0.090,Y -269.379,Z 888.327,A 0.000,B 0.000,C 90.000,E1 58.869} C_DIS
LIN {X 0.013,Y -257.085,Z 888.309,A 0.000,B 0.000,C 90.000,E1 55.674} C_DIS
LIN {X -0.011,Y -245.876,Z 888.291,A 0.000,B 0.000,C 90.000,E1 52.431} C_DIS
LIN {X 0.073,Y -235.958,Z 888.273,A 0.000,B 0.000,C 90.000,E1 49.094} C_DIS
LIN {X -0.086,Y -227.852,Z 888.256,A 0.000,B 0.000,C 90.000,E1 46.134} C_DIS
LIN {X 0.030,Y -218.326,Z 888.235,A 0.000,B 0.000,C 90.000,E1 42.285} C_DIS
LIN {X -0.051,Y -211.241,Z 888.218,A 0.000,B 0.000,C 90.000,E1 39.197} C_DIS
LIN {X 0.051,Y -204.565,Z 888.200,A 0.000,B 0.000,C 90.000,E1 36.011} C_DIS
LIN {X -0.035,Y -198.380,Z 888.182,A 0.000,B 0.000,C 90.000,E1 32.832} C_DIS
LIN {X -0.046,Y -192.748,Z 888.164,A 0.000,B 0.000,C 90.000,E1 29.589} C_DIS
LIN {X 0.014,Y -187.742,Z 888.146,A 0.000,B 0.000,C 90.000,E1 26.283} C_DIS
LIN {X 0.044,Y -183.436,Z 888.128,A 0.000,B 0.000,C 90.000,E1 22.950} C_DIS
LIN {X -0.071,Y -179.779,Z 888.109,A 0.000,B 0.000,C 90.000,E1 19.631} C_DIS
LIN {X 0.013,Y -176.272,Z 888.085,A 0.000,B 0.000,C 90.000,E1 15.371} C_DIS
LIN {X -0.001,Y -173.489,Z 888.057,A 0.000,B 0.000,C 90.000,E1 10.254} C_DIS
LIN {X 0.013,Y -174.328,Z 887.964,A 0.000,B 0.000,C 90.000,E1 353.514} C_DIS
LIN {X 0.079,Y -176.993,Z 887.940,A 0.000,B 0.000,C 90.000,E1 349.218} C_DIS
LIN {X 0.021,Y -180.686,Z 887.917,A 0.000,B 0.000,C 90.000,E1 344.991} C_DIS
LIN {X -0.032,Y -184.536,Z 887.898,A 0.000,B 0.000,C 90.000,E1 341.638} C_DIS
LIN {X 0.015,Y -189.190,Z 887.879,A 0.000,B 0.000,C 90.000,E1 338.284} C_DIS
LIN {X 0.040,Y -194.561,Z 887.861,A 0.000,B 0.000,C 90.000,E1 334.973} C_DIS
LIN {X -0.042,Y -202.080,Z 887.838,A 0.000,B 0.000,C 90.000,E1 330.923} C_DIS
LIN {X -0.028,Y -210.180,Z 887.816,A 0.000,B 0.000,C 90.000,E1 326.914} C_DIS
LIN {X 0.014,Y -217.161,Z 887.799,A 0.000,B 0.000,C 90.000,E1 323.749} C_DIS
LIN {X -0.052,Y -225.733,Z 887.779,A 0.000,B 0.000,C 90.000,E1 320.275} C_DIS
LIN {X -0.047,Y -234.112,Z 887.762,A 0.000,B 0.000,C 90.000,E1 317.229} C_DIS
LIN {X -0.036,Y -244.784,Z 887.744,A 0.000,B 0.000,C 90.000,E1 313.866} C_DIS
LIN {X 0.144,Y -256.664,Z 887.725,A 0.000,B 0.000,C 90.000,E1 310.539} C_DIS
LIN {X 0.002,Y -269.828,Z 887.708,A 0.000,B 0.000,C 90.000,E1 307.363} C_DIS
LIN {X -0.044,Y -284.135,Z 887.690,A 0.000,B 0.000,C 90.000,E1 304.246} C_DIS
LIN {X -0.075,Y -299.860,Z 887.673,A 0.000,B 0.000,C 90.000,E1 301.209} C_DIS
LIN {X 0.063,Y -317.244,Z 887.657,A 0.000,B 0.000,C 90.000,E1 298.231} C_DIS
LIN {X 0.088,Y -330.016,Z 887.646,A 0.000,B 0.000,C 90.000,E1 296.309} C_DIS
LIN {X -0.041,Y -343.881,Z 887.636,A 0.000,B 0.000,C 90.000,E1 294.463} C_DIS
LIN {X 0.039,Y -363.588,Z 887.622,A 0.000,B 0.000,C 90.000,E1 292.025} C_DIS
LIN {X -0.026,Y -381.701,Z 887.611,A 0.000,B 0.000,C 90.000,E1 289.993} C_DIS
LIN {X -0.167,Y -402.377,Z 887.599,A 0.000,B 0.000,C 90.000,E1 287.819} C_DIS
LIN {X 0.122,Y -415.153,Z 887.591,A 0.000,B 0.000,C 90.000,E1 286.441} C_DIS
LIN {X 0.108,Y -425.156,Z 887.585,A 0.000,B 0.000,C 90.000,E1 285.371} C_DIS
LIN {X -0.175,Y -437.255,Z 887.578,A 0.000,B 0.000,C 90.000,E1 284.064} C_DIS
LIN {X -0.210,Y -446.411,Z 887.572,A 0.000,B 0.000,C 90.000,E1 283.008} C_DIS
LIN {X -0.135,Y -455.117,Z 887.566,A 0.000,B 0.000,C 90.000,E1 281.951} C_DIS
LIN {X 0.045,Y -463.186,Z 887.561,A 0.000,B 0.000,C 90.000,E1 280.894} C_DIS
LIN {X -0.228,Y -470.691,Z 887.555,A 0.000,B 0.000,C 90.000,E1 279.905} C_DIS
LIN {X 0.192,Y -475.891,Z 887.551,A 0.000,B 0.000,C 90.000,E1 279.095} C_DIS
LIN {X 0.188,Y -480.519,Z 887.546,A 0.000,B 0.000,C 90.000,E1 278.341} C_DIS
LIN {X -0.064,Y -483.241,Z 887.544,A 0.000,B 0.000,C 90.000,E1 277.871} C_DIS
LIN {X -0.069,Y -486.683,Z 887.540,A 0.000,B 0.000,C 90.000,E1 277.125} C_DIS
LIN {X -0.186,Y -487.706,Z 887.538,A 0.000,B 0.000,C 90.000,E1 276.891} C_DIS
LIN {X 0.016,Y -489.401,Z 887.535,A 0.000,B 0.000,C 90.000,E1 276.372} C_DIS
LIN {X 0.227,Y -490.807,Z 887.533,A 0.000,B 0.000,C 90.000,E1 275.853} C_DIS
LIN {X -0.043,Y -491.840,Z 887.530,A 0.000,B 0.000,C 90.000,E1 275.391} C_DIS
LIN {X 0.140,Y -492.479,Z 887.527,A 0.000,B 0.000,C 90.000,E1 274.878} C_DIS
LIN {X -0.117,Y -492.723,Z 887.524,A 0.000,B 0.000,C 90.000,E1 274.416} C_DIS
LIN {X 0.117,Y -492.462,Z 887.522,A 0.000,B 0.000,C 90.000,E1 273.898} C_DIS
LIN {X -0.171,Y -491.833,Z 887.519,A 0.000,B 0.000,C 90.000,E1 273.440} C_DIS
LIN {X 0.060,Y -490.756,Z 887.516,A 0.000,B 0.000,C 90.000,E1 272.922} C_DIS
LIN {X -0.228,Y -489.211,Z 887.514,A 0.000,B 0.000,C 90.000,E1 272.465} C_DIS
LIN {X -0.030,Y -487.111,Z 887.511,A 0.000,B 0.000,C 90.000,E1 271.949} C_DIS
LIN {X 0.173,Y -484.366,Z 887.508,A 0.000,B 0.000,C 90.000,E1 271.432} C_DIS
LIN {X 0.014,Y -482.784,Z 887.507,A 0.000,B 0.000,C 90.000,E1 271.203} C_DIS
LIN {X 0.172,Y -478.925,Z 887.504,A 0.000,B 0.000,C 90.000,E1 270.688} C_DIS
LIN {X 0.009,Y -476.699,Z 887.503,A 0.000,B 0.000,C 90.000,E1 270.458} C_DIS
LIN {X 0.136,Y -471.515,Z 887.500,A 0.000,B 0.000,C 90.000,E1 269.943} C_DIS
LIN {X -0.044,Y -465.390,Z 887.497,A 0.000,B 0.000,C 90.000,E1 269.484} C_DIS
LIN {X 0.148,Y -462.407,Z 887.496,A 0.000,B 0.000,C 90.000,E1 269.255} C_DIS
LIN {X -0.140,Y -455.870,Z 887.494,A 0.000,B 0.000,C 90.000,E1 268.912} C_DIS
LIN {X 0.030,Y -449.049,Z 887.492,A 0.000,B 0.000,C 90.000,E1 268.568} C_DIS
LIN {X 0.108,Y -441.925,Z 887.491,A 0.000,B 0.000,C 90.000,E1 268.282} C_DIS
LIN {X 0.153,Y -434.172,Z 887.489,A 0.000,B 0.000,C 90.000,E1 268.051} C_DIS
LIN {X 0.165,Y -426.362,Z 887.488,A 0.000,B 0.000,C 90.000,E1 267.879} C_DIS
LIN {X 0.085,Y -417.497,Z 887.488,A 0.000,B 0.000,C 90.000,E1 267.764} C_DIS
LIN {X 0.120,Y -410.470,Z 887.487,A 0.000,B 0.000,C 90.000,E1 267.707} C_DIS
LIN {X 0.029,Y -181.081,Z 887.487,A 0.000,B 0.000,C 90.000,E1 267.707} C_DIS
LIN {X 0.036,Y -180.887,Z 887.473,A 0.000,B 0.000,C 90.000,E1 265.122} C_DIS
LIN {X -0.082,Y -179.009,Z 887.445,A 0.000,B 0.000,C 90.000,E1 260.095} C_DIS
LIN {X 0.013,Y -178.623,Z 887.440,A 0.000,B 0.000,C 90.000,E1 259.218} C_DIS
LIN {X -0.088,Y -175.674,Z 887.412,A 0.000,B 0.000,C 90.000,E1 254.157} C_DIS
LIN {X -0.076,Y -172.391,Z 887.388,A 0.000,B 0.000,C 90.000,E1 249.880} C_DIS
LIN {X -0.060,Y -171.196,Z 887.379,A 0.000,B 0.000,C 90.000,E1 248.156} C_DIS
LIN {X -0.008,Y -167.485,Z 887.355,A 0.000,B 0.000,C 90.000,E1 243.819} C_DIS
LIN {X 0.000,Y -166.882,Z 887.350,A 0.000,B 0.000,C 90.000,E1 242.948} C_DIS
LIN {X -0.009,Y -162.187,Z 887.321,A 0.000,B 0.000,C 90.000,E1 237.709} C_DIS
LIN {X -0.042,Y -160.756,Z 887.311,A 0.000,B 0.000,C 90.000,E1 235.960} C_DIS
LIN {X 0.027,Y -157.553,Z 887.291,A 0.000,B 0.000,C 90.000,E1 232.396} C_DIS
LIN {X -0.035,Y -155.582,Z 887.276,A 0.000,B 0.000,C 90.000,E1 229.747} C_DIS
LIN {X 0.017,Y -151.866,Z 887.251,A 0.000,B 0.000,C 90.000,E1 225.243} C_DIS
LIN {X 0.030,Y -150.090,Z 887.236,A 0.000,B 0.000,C 90.000,E1 222.528} C_DIS
LIN {X -0.052,Y -146.891,Z 887.211,A 0.000,B 0.000,C 90.000,E1 218.016} C_DIS
LIN {X 0.053,Y -145.478,Z 887.196,A 0.000,B 0.000,C 90.000,E1 215.231} C_DIS
LIN {X -0.031,Y -142.888,Z 887.170,A 0.000,B 0.000,C 90.000,E1 210.669} C_DIS
LIN {X 0.026,Y -141.507,Z 887.150,A 0.000,B 0.000,C 90.000,E1 206.950} C_DIS
LIN {X -0.056,Y -139.391,Z 887.114,A 0.000,B 0.000,C 90.000,E1 200.482} C_DIS
LIN {X -0.005,Y -139.098,Z 887.103,A 0.000,B 0.000,C 90.000,E1 198.598} C_DIS
LIN {X -0.013,Y -138.353,Z 887.057,A 0.000,B 0.000,C 90.000,E1 190.197} C_DIS
LIN {X -0.020,Y -139.515,Z 887.005,A 0.000,B 0.000,C 90.000,E1 180.859} C_DIS
LIN {X 0.061,Y -141.167,Z 886.974,A 0.000,B 0.000,C 90.000,E1 175.241} C_DIS
LIN {X 0.032,Y -142.546,Z 886.958,A 0.000,B 0.000,C 90.000,E1 172.470} C_DIS
LIN {X -0.042,Y -144.821,Z 886.933,A 0.000,B 0.000,C 90.000,E1 167.881} C_DIS
LIN {X -0.055,Y -147.442,Z 886.912,A 0.000,B 0.000,C 90.000,E1 164.212} C_DIS
LIN {X -0.027,Y -150.023,Z 886.892,A 0.000,B 0.000,C 90.000,E1 160.550} C_DIS
LIN {X -0.021,Y -153.358,Z 886.872,A 0.000,B 0.000,C 90.000,E1 156.922} C_DIS
LIN {X 0.027,Y -155.892,Z 886.857,A 0.000,B 0.000,C 90.000,E1 154.204} C_DIS
LIN {X -0.075,Y -159.750,Z 886.837,A 0.000,B 0.000,C 90.000,E1 150.667} C_DIS
LIN {X -0.009,Y -161.990,Z 886.827,A 0.000,B 0.000,C 90.000,E1 148.869} C_DIS
LIN {X 0.011,Y -166.182,Z 886.807,A 0.000,B 0.000,C 90.000,E1 145.341} C_DIS
LIN {X 0.004,Y -171.198,Z 886.788,A 0.000,B 0.000,C 90.000,E1 141.859} C_DIS
LIN {X 0.034,Y -176.080,Z 886.769,A 0.000,B 0.000,C 90.000,E1 138.405} C_DIS
LIN {X -0.104,Y -180.340,Z 886.755,A 0.000,B 0.000,C 90.000,E1 135.891} C_DIS
LIN {X 0.005,Y -185.750,Z 886.736,A 0.000,B 0.000,C 90.000,E1 132.486} C_DIS
LIN {X -0.082,Y -190.362,Z 886.722,A 0.000,B 0.000,C 90.000,E1 130.011} C_DIS
LIN {X -0.023,Y -193.307,Z 886.713,A 0.000,B 0.000,C 90.000,E1 128.257} C_DIS
LIN {X -0.071,Y -294.668,Z 886.712,A 0.000,B 0.000,C 90.000,E1 128.257} C_DIS
LIN {X 0.101,Y -297.086,Z 886.712,A 0.000,B 0.000,C 90.000,E1 128.177} C_DIS
LIN {X -0.008,Y -302.748,Z 886.710,A 0.000,B 0.000,C 90.000,E1 127.855} C_DIS
LIN {X -0.066,Y -305.764,Z 886.708,A 0.000,B 0.000,C 90.000,E1 127.523} C_DIS
LIN {X -0.013,Y -307.749,Z 886.707,A 0.000,B 0.000,C 90.000,E1 127.202} C_DIS
LIN {X 0.100,Y -309.300,Z 886.705,A 0.000,B 0.000,C 90.000,E1 126.870} C_DIS
LIN {X -0.116,Y -310.584,Z 886.703,A 0.000,B 0.000,C 90.000,E1 126.583} C_DIS
LIN {X 0.097,Y -322.897,Z 886.682,A 0.000,B 0.000,C 90.000,E1 122.673} C_DIS
LIN {X -0.163,Y -333.546,Z 886.666,A 0.000,B 0.000,C 90.000,E1 119.873} C_DIS
LIN {X 0.007,Y -345.561,Z 886.650,A 0.000,B 0.000,C 90.000,E1 117.052} C_DIS
LIN {X -0.108,Y -359.053,Z 886.635,A 0.000,B 0.000,C 90.000,E1 114.335} C_DIS
LIN {X -0.078,Y -372.380,Z 886.622,A 0.000,B 0.000,C 90.000,E1 111.950} C_DIS
LIN {X -0.137,Y -387.062,Z 886.609,A 0.000,B 0.000,C 90.000,E1 109.631} C_DIS
LIN {X 0.048,Y -403.204,Z 886.596,A 0.000,B 0.000,C 90.000,E1 107.330} C_DIS
LIN {X -0.105,Y -420.922,Z 886.584,A 0.000,B 0.000,C 90.000,E1 105.134} C_DIS
LIN {X 0.134,Y -440.283,Z 886.572,A 0.000,B 0.000,C 90.000,E1 102.952} C_DIS
LIN {X 0.161,Y -460.495,Z 886.561,A 0.000,B 0.000,C 90.000,E1 100.950} C_DIS
LIN {X 0.096,Y -468.043,Z 886.557,A 0.000,B 0.000,C 90.000,E1 100.254} C_DIS
LIN {X 0.130,Y -469.883,Z 886.556,A 0.000,B 0.000,C 90.000,E1 100.018} C_DIS
LIN {X -0.101,Y -471.412,Z 886.554,A 0.000,B 0.000,C 90.000,E1 99.792} C_DIS
LIN {X 0.215,Y -472.555,Z 886.553,A 0.000,B 0.000,C 90.000,E1 99.500} C_DIS
LIN {X -0.070,Y -473.929,Z 886.550,A 0.000,B 0.000,C 90.000,E1 99.029} C_DIS
LIN {X 0.043,Y -474.280,Z 886.547,A 0.000,B 0.000,C 90.000,E1 98.511} C_DIS
LIN {X 0.166,Y -473.670,Z 886.544,A 0.000,B 0.000,C 90.000,E1 97.992} C_DIS
LIN {X -0.174,Y -472.002,Z 886.542,A 0.000,B 0.000,C 90.000,E1 97.530} C_DIS
LIN {X 0.152,Y -470.681,Z 886.540,A 0.000,B 0.000,C 90.000,E1 97.239} C_DIS
LIN {X 0.068,Y -454.689,Z 886.526,A 0.000,B 0.000,C 90.000,E1 94.702} C_DIS
LIN {X 0.226,Y -444.190,Z 886.516,A 0.000,B 0.000,C 90.000,E1 92.865} C_DIS
LIN {X -0.181,Y -436.357,Z 886.509,A 0.000,B 0.000,C 90.000,E1 91.604} C_DIS
LIN {X -0.124,Y -426.791,Z 886.500,A 0.000,B 0.000,C 90.000,E1 90.000} C_DIS
LIN {X -0.115,Y -415.390,Z 886.489,A 0.000,B 0.000,C 90.000,E1 88.108} C_DIS
LIN {X 0.061,Y -404.070,Z 886.479,A 0.000,B 0.000,C 90.000,E1 86.159} C_DIS
LIN {X 0.107,Y -391.206,Z 886.466,A 0.000,B 0.000,C 90.000,E1 83.913} C_DIS
LIN {X -0.119,Y -380.106,Z 886.455,A 0.000,B 0.000,C 90.000,E1 81.951} C_DIS
LIN {X -0.156,Y -368.929,Z 886.444,A 0.000,B 0.000,C 90.000,E1 79.926} C_DIS
LIN {X 0.055,Y -357.801,Z 886.432,A 0.000,B 0.000,C 90.000,E1 77.825} C_DIS
LIN {X -0.095,Y -348.139,Z 886.422,A 0.000,B 0.000,C 90.000,E1 76.047} C_DIS
LIN {X 0.031,Y -333.906,Z 886.407,A 0.000,B 0.000,C 90.000,E1 73.268} C_DIS
LIN {X 0.144,Y -320.285,Z 886.391,A 0.000,B 0.000,C 90.000,E1 70.423} C_DIS
LIN {X -0.133,Y -309.988,Z 886.379,A 0.000,B 0.000,C 90.000,E1 68.230} C_DIS
LIN {X -0.108,Y -298.431,Z 886.364,A 0.000,B 0.000,C 90.000,E1 65.613} C_DIS
LIN {X 0.026,Y -288.254,Z 886.351,A 0.000,B 0.000,C 90.000,E1 63.256} C_DIS
LIN {X -0.146,Y -279.533,Z 886.340,A 0.000,B 0.000,C 90.000,E1 61.257} C_DIS
LIN {X 0.101,Y -269.429,Z 886.327,A 0.000,B 0.000,C 90.000,E1 58.791} C_DIS
LIN {X -0.156,Y -257.192,Z 886.309,A 0.000,B 0.000,C 90.000,E1 55.674} C_DIS
LIN {X -0.020,Y -246.052,Z 886.291,A 0.000,B 0.000,C 90.000,E1 52.396} C_DIS
LIN {X -0.075,Y -236.147,Z 886.273,A 0.000,B 0.000,C 90.000,E1 49.094} C_DIS
LIN {X -0.014,Y -226.109,Z 886.252,A 0.000,B 0.000,C 90.000,E1 45.324} C_DIS
LIN {X 0.066,Y -218.541,Z 886.235,A 0.000,B 0.000,C 90.000,E1 42.243} C_DIS
LIN {X -0.004,Y -211.462,Z 886.218,A 0.000,B 0.000,C 90.000,E1 39.152} C_DIS
LIN {X -0.056,Y -204.778,Z 886.200,A 0.000,B 0.000,C 90.000,E1 36.011} C_DIS
LIN {X -0.026,Y -198.595,Z 886.182,A 0.000,B 0.000,C 90.000,E1 32.801} C_DIS
LIN {X 0.030,Y -192.970,Z 886.164,A 0.000,B 0.000,C 90.000,E1 29.539} C_DIS
LIN {X 0.100,Y -187.963,Z 886.146,A 0.000,B 0.000,C 90.000,E1 26.232} C_DIS
LIN {X -0.032,Y -183.654,Z 886.127,A 0.000,B 0.000,C 90.000,E1 22.950} C_DIS
LIN {X 0.029,Y -180.021,Z 886.109,A 0.000,B 0.000,C 90.000,E1 19.577} C_DIS
LIN {X -0.048,Y -176.517,Z 886.085,A 0.000,B 0.000,C 90.000,E1 15.371} C_DIS
LIN {X -0.051,Y -173.761,Z 886.057,A 0.000,B 0.000,C 90.000,E1 10.254} C_DIS
LIN {X 0.027,Y -174.632,Z 885.964,A 0.000,B 0.000,C 90.000,E1 353.514} C_DIS
LIN {X 0.102,Y -177.306,Z 885.940,A 0.000,B 0.000,C 90.000,E1 349.218} C_DIS
LIN {X 0.054,Y -181.034,Z 885.917,A 0.000,B 0.000,C 90.000,E1 344.991} C_DIS
LIN {X 0.011,Y -184.903,Z 885.898,A 0.000,B 0.000,C 90.000,E1 341.638} C_DIS
LIN {X 0.068,Y -189.555,Z 885.879,A 0.000,B 0.000,C 90.000,E1 338.284} C_DIS
LIN {X 0.104,Y -194.937,Z 885.861,A 0.000,B 0.000,C 90.000,E1 334.973} C_DIS
LIN {X 0.036,Y -202.440,Z 885.839,A 0.000,B 0.000,C 90.000,E1 330.923} C_DIS
LIN {X 0.065,Y -210.480,Z 885.816,A 0.000,B 0.000,C 90.000,E1 326.914} C_DIS
LIN {X -0.012,Y -217.459,Z 885.799,A 0.000,B 0.000,C 90.000,E1 323.783} C_DIS
LIN {X 0.065,Y -226.015,Z 885.779,A 0.000,B 0.000,C 90.000,E1 320.275} C_DIS
LIN {X 0.074,Y -234.373,Z 885.763,A 0.000,B 0.000,C 90.000,E1 317.229} C_DIS
LIN {X 0.098,Y -245.040,Z 885.744,A 0.000,B 0.000,C 90.000,E1 313.866} C_DIS
LIN {X -0.070,Y -256.888,Z 885.726,A 0.000,B 0.000,C 90.000,E1 310.620} C_DIS
LIN {X -0.002,Y -269.972,Z 885.708,A 0.000,B 0.000,C 90.000,E1 307.397} C_DIS
LIN {X -0.030,Y -284.209,Z 885.690,A 0.000,B 0.000,C 90.000,E1 304.278} C_DIS
LIN {X 0.109,Y -299.853,Z 885.674,A 0.000,B 0.000,C 90.000,E1 301.209} C_DIS
LIN {X -0.022,Y -317.150,Z 885.657,A 0.000,B 0.000,C 90.000,E1 298.281} C_DIS
LIN {X -0.008,Y -329.855,Z 885.646,A 0.000,B 0.000,C 90.000,E1 296.360} C_DIS
LIN {X -0.137,Y -346.033,Z 885.634,A 0.000,B 0.000,C 90.000,E1 294.207} C_DIS
LIN {X 0.020,Y -368.368,Z 885.619,A 0.000,B 0.000,C 90.000,E1 291.461} C_DIS
LIN {X -0.178,Y -383.867,Z 885.610,A 0.000,B 0.000,C 90.000,E1 289.758} C_DIS
LIN {X 0.011,Y -401.932,Z 885.599,A 0.000,B 0.000,C 90.000,E1 287.819} C_DIS
LIN {X -0.008,Y -414.663,Z 885.592,A 0.000,B 0.000,C 90.000,E1 286.496} C_DIS
LIN {X -0.018,Y -424.663,Z 885.586,A 0.000,B 0.000,C 90.000,E1 285.426} C_DIS
LIN {X 0.102,Y -436.815,Z 885.578,A 0.000,B 0.000,C 90.000,E1 284.064} C_DIS
LIN {X -0.140,Y -448.217,Z 885.571,A 0.000,B 0.000,C 90.000,E1 282.771} C_DIS
LIN {X -0.042,Y -456.847,Z 885.565,A 0.000,B 0.000,C 90.000,E1 281.715} C_DIS
LIN {X 0.157,Y -464.811,Z 885.559,A 0.000,B 0.000,C 90.000,E1 280.658} C_DIS
LIN {X -0.098,Y -472.187,Z 885.554,A 0.000,B 0.000,C 90.000,E1 279.670} C_DIS
LIN {X -0.141,Y -477.253,Z 885.549,A 0.000,B 0.000,C 90.000,E1 278.916} C_DIS
LIN {X -0.134,Y -481.723,Z 885.545,A 0.000,B 0.000,C 90.000,E1 278.163} C_DIS
LIN {X -0.093,Y -485.468,Z 885.541,A 0.000,B 0.000,C 90.000,E1 277.409} C_DIS
LIN {X 0.094,Y -487.570,Z 885.538,A 0.000,B 0.000,C 90.000,E1 276.891} C_DIS
LIN {X -0.189,Y -489.331,Z 885.536,A 0.000,B 0.000,C 90.000,E1 276.429} C_DIS
LIN {X 0.019,Y -490.727,Z 885.533,A 0.000,B 0.000,C 90.000,E1 275.910} C_DIS
LIN {X 0.237,Y -491.801,Z 885.530,A 0.000,B 0.000,C 90.000,E1 275.391} C_DIS
LIN {X -0.071,Y -492.511,Z 885.527,A 0.000,B 0.000,C 90.000,E1 274.935} C_DIS
LIN {X 0.163,Y -492.742,Z 885.525,A 0.000,B 0.000,C 90.000,E1 274.416} C_DIS
LIN {X -0.093,Y -492.598,Z 885.522,A 0.000,B 0.000,C 90.000,E1 273.955} C_DIS
LIN {X 0.110,Y -491.992,Z 885.519,A 0.000,B 0.000,C 90.000,E1 273.440} C_DIS
LIN {X -0.149,Y -490.975,Z 885.516,A 0.000,B 0.000,C 90.000,E1 272.980} C_DIS
LIN {X 0.053,Y -489.477,Z 885.514,A 0.000,B 0.000,C 90.000,E1 272.465} C_DIS
LIN {X -0.237,Y -487.427,Z 885.511,A 0.000,B 0.000,C 90.000,E1 272.007} C_DIS
LIN {X -0.032,Y -484.772,Z 885.508,A 0.000,B 0.000,C 90.000,E1 271.489} C_DIS
LIN {X 0.138,Y -481.440,Z 885.505,A 0.000,B 0.000,C 90.000,E1 270.974} C_DIS
LIN {X -0.188,Y -477.314,Z 885.503,A 0.000,B 0.000,C 90.000,E1 270.516} C_DIS
LIN {X -0.055,Y -472.192,Z 885.500,A 0.000,B 0.000,C 90.000,E1 270.000} C_DIS
LIN {X -0.168,Y -466.417,Z 885.497,A 0.000,B 0.000,C 90.000,E1 269.542} C_DIS
LIN {X 0.133,Y -460.136,Z 885.495,A 0.000,B 0.000,C 90.000,E1 269.083} C_DIS
LIN {X -0.021,Y -453.422,Z 885.493,A 0.000,B 0.000,C 90.000,E1 268.740} C_DIS
LIN {X -0.151,Y -446.556,Z 885.491,A 0.000,B 0.000,C 90.000,E1 268.453} C_DIS
LIN {X 0.083,Y -439.060,Z 885.490,A 0.000,B 0.000,C 90.000,E1 268.165} C_DIS
LIN {X -0.142,Y -431.257,Z 885.489,A 0.000,B 0.000,C 90.000,E1 267.993} C_DIS
LIN {X -0.002,Y -423.051,Z 885.488,A 0.000,B 0.000,C 90.000,E1 267.822} C_DIS
LIN {X -0.187,Y -416.088,Z 885.487,A 0.000,B 0.000,C 90.000,E1 267.764} C_DIS
LIN {X -0.079,Y -408.609,Z 885.487,A 0.000,B 0.000,C 90.000,E1 267.707} C_DIS
LIN {X -0.060,Y -181.076,Z 885.487,A 0.000,B 0.000,C 90.000,E1 267.707} C_DIS
LIN {X 0.001,Y -180.885,Z 885.473,A 0.000,B 0.000,C 90.000,E1 265.122} C_DIS
LIN {X 0.060,Y -179.006,Z 885.445,A 0.000,B 0.000,C 90.000,E1 260.038} C_DIS
LIN {X -0.022,Y -178.615,Z 885.440,A 0.000,B 0.000,C 90.000,E1 259.218} C_DIS
LIN {X 0.047,Y -175.666,Z 885.412,A 0.000,B 0.000,C 90.000,E1 254.102} C_DIS
LIN {X 0.051,Y -172.384,Z 885.388,A 0.000,B 0.000,C 90.000,E1 249.826} C_DIS
LIN {X 0.065,Y -171.184,Z 885.378,A 0.000,B 0.000,C 90.000,E1 248.103} C_DIS
LIN {X -0.042,Y -167.476,Z 885.354,A 0.000,B 0.000,C 90.000,E1 243.819} C_DIS
LIN {X -0.034,Y -166.873,Z 885.350,A 0.000,B 0.000,C 90.000,E1 242.948} C_DIS
LIN {X -0.042,Y -162.178,Z 885.320,A 0.000,B 0.000,C 90.000,E1 237.709} C_DIS
LIN {X 0.016,Y -160.744,Z 885.311,A 0.000,B 0.000,C 90.000,E1 235.928} C_DIS
LIN {X -0.006,Y -157.544,Z 885.291,A 0.000,B 0.000,C 90.000,E1 232.396} C_DIS
LIN {X -0.067,Y -155.571,Z 885.276,A 0.000,B 0.000,C 90.000,E1 229.747} C_DIS
LIN {X -0.015,Y -151.858,Z 885.251,A 0.000,B 0.000,C 90.000,E1 225.243} C_DIS
LIN {X -0.001,Y -150.080,Z 885.236,A 0.000,B 0.000,C 90.000,E1 222.528} C_DIS
LIN {X 0.032,Y -146.884,Z 885.211,A 0.000,B 0.000,C 90.000,E1 217.971} C_DIS
LIN {X 0.022,Y -145.471,Z 885.196,A 0.000,B 0.000,C 90.000,E1 215.231} C_DIS
LIN {X -0.062,Y -142.883,Z 885.170,A 0.000,B 0.000,C 90.000,E1 210.669} C_DIS
LIN {X -0.005,Y -141.501,Z 885.150,A 0.000,B 0.000,C 90.000,E1 206.950} C_DIS
LIN {X 0.044,Y -139.389,Z 885.114,A 0.000,B 0.000,C 90.000,E1 200.429} C_DIS
LIN {X 0.033,Y -138.846,Z 885.098,A 0.000,B 0.000,C 90.000,E1 197.638} C_DIS
LIN {X -0.043,Y -138.354,Z 885.057,A 0.000,B 0.000,C 90.000,E1 190.197} C_DIS
LIN {X -0.051,Y -139.517,Z 885.005,A 0.000,B 0.000,C 90.000,E1 180.859} C_DIS
LIN {X 0.030,Y -141.172,Z 884.974,A 0.000,B 0.000,C 90.000,E1 175.241} C_DIS
LIN {X 0.001,Y -142.551,Z 884.958,A 0.000,B 0.000,C 90.000,E1 172.470} C_DIS
LIN {X -0.073,Y -144.829,Z 884.932,A 0.000,B 0.000,C 90.000,E1 167.881} C_DIS
LIN {X 0.055,Y -147.451,Z 884.912,A 0.000,B 0.000,C 90.000,E1 164.157} C_DIS
LIN {X -0.059,Y -150.032,Z 884.892,A 0.000,B 0.000,C 90.000,E1 160.550} C_DIS
LIN {X -0.053,Y -153.371,Z 884.872,A 0.000,B 0.000,C 90.000,E1 156.922} C_DIS
LIN {X -0.005,Y -155.903,Z 884.857,A 0.000,B 0.000,C 90.000,E1 154.204} C_DIS
LIN {X -0.028,Y -159.765,Z 884.837,A 0.000,B 0.000,C 90.000,E1 150.639} C_DIS
LIN {X -0.041,Y -162.005,Z 884.827,A 0.000,B 0.000,C 90.000,E1 148.869} C_DIS
LIN {X 0.072,Y -166.198,Z 884.807,A 0.000,B 0.000,C 90.000,E1 145.308} C_DIS
LIN {X 0.075,Y -171.214,Z 884.788,A 0.000,B 0.000,C 90.000,E1 141.823} C_DIS
LIN {X -0.001,Y -176.097,Z 884.769,A 0.000,B 0.000,C 90.000,E1 138.405} C_DIS
LIN {X 0.116,Y -180.360,Z 884.755,A 0.000,B 0.000,C 90.000,E1 135.810} C_DIS
LIN {X 0.093,Y -185.769,Z 884.736,A 0.000,B 0.000,C 90.000,E1 132.447} C_DIS
LIN {X 0.027,Y -190.383,Z 884.722,A 0.000,B 0.000,C 90.000,E1 129.967} C_DIS
LIN {X 0.021,Y -193.285,Z 884.713,A 0.000,B 0.000,C 90.000,E1 128.257} C_DIS
LIN {X -0.021,Y -294.896,Z 884.713,A 0.000,B 0.000,C 90.000,E1 128.257} C_DIS
LIN {X -0.164,Y -300.118,Z 884.711,A 0.000,B 0.000,C 90.000,E1 128.096} C_DIS
LIN {X -0.072,Y -302.582,Z 884.710,A 0.000,B 0.000,C 90.000,E1 127.890} C_DIS
LIN {X -0.124,Y -305.881,Z 884.708,A 0.000,B 0.000,C 90.000,E1 127.523} C_DIS
LIN {X 0.168,Y -307.832,Z 884.707,A 0.000,B 0.000,C 90.000,E1 127.156} C_DIS
LIN {X 0.029,Y -309.358,Z 884.705,A 0.000,B 0.000,C 90.000,E1 126.870} C_DIS
LIN {X -0.187,Y -310.618,Z 884.703,A 0.000,B 0.000,C 90.000,E1 126.583} C_DIS
LIN {X -0.059,Y -321.818,Z 884.683,A 0.000,B 0.000,C 90.000,E1 123.007} C_DIS
LIN {X 0.101,Y -332.324,Z 884.667,A 0.000,B 0.000,C 90.000,E1 120.129} C_DIS
LIN {X 0.080,Y -344.192,Z 884.652,A 0.000,B 0.000,C 90.000,E1 117.334} C_DIS
LIN {X 0.096,Y -357.517,Z 884.637,A 0.000,B 0.000,C 90.000,E1 114.591} C_DIS
LIN {X 0.099,Y -370.688,Z 884.623,A 0.000,B 0.000,C 90.000,E1 112.206} C_DIS
LIN {X 0.011,Y -385.202,Z 884.610,A 0.000,B 0.000,C 90.000,E1 109.885} C_DIS
LIN {X 0.164,Y -401.162,Z 884.598,A 0.000,B 0.000,C 90.000,E1 107.583} C_DIS
LIN {X 0.088,Y -418.683,Z 884.585,A 0.000,B 0.000,C 90.000,E1 105.371} C_DIS
LIN {X -0.172,Y -437.863,Z 884.573,A 0.000,B 0.000,C 90.000,E1 103.244} C_DIS
LIN {X 0.123,Y -458.006,Z 884.562,A 0.000,B 0.000,C 90.000,E1 101.186} C_DIS
LIN {X 0.014,Y -468.111,Z 884.557,A 0.000,B 0.000,C 90.000,E1 100.254} C_DIS
LIN {X 0.047,Y -469.935,Z 884.556,A 0.000,B 0.000,C 90.000,E1 100.018} C_DIS
LIN {X -0.183,Y -471.452,Z 884.554,A 0.000,B 0.000,C 90.000,E1 99.792} C_DIS
LIN {X 0.132,Y -472.587,Z 884.553,A 0.000,B 0.000,C 90.000,E1 99.500} C_DIS
LIN {X -0.152,Y -473.946,Z 884.550,A 0.000,B 0.000,C 90.000,E1 99.029} C_DIS
LIN {X -0.039,Y -474.285,Z 884.547,A 0.000,B 0.000,C 90.000,E1 98.511} C_DIS
LIN {X 0.085,Y -473.661,Z 884.544,A 0.000,B 0.000,C 90.000,E1 97.992} C_DIS
LIN {X -0.256,Y -471.978,Z 884.542,A 0.000,B 0.000,C 90.000,E1 97.530} C_DIS
LIN {X 0.071,Y -470.646,Z 884.540,A 0.000,B 0.000,C 90.000,E1 97.239} C_DIS
LIN {X 0.183,Y -456.179,Z 884.528,A 0.000,B 0.000,C 90.000,E1 94.935} C_DIS
LIN {X 0.148,Y -444.158,Z 884.516,A 0.000,B 0.000,C 90.000,E1 92.865} C_DIS
LIN {X 0.177,Y -436.324,Z 884.509,A 0.000,B 0.000,C 90.000,E1 91.547} C_DIS
LIN {X -0.201,Y -426.783,Z 884.500,A 0.000,B 0.000,C 90.000,E1 90.000} C_DIS
LIN {X -0.190,Y -415.360,Z 884.489,A 0.000,B 0.000,C 90.000,E1 88.108} C_DIS
LIN {X -0.012,Y -404.032,Z 884.479,A 0.000,B 0.000,C 90.000,E1 86.159} C_DIS
LIN {X -0.021,Y -392.758,Z 884.468,A 0.000,B 0.000,C 90.000,E1 84.204} C_DIS
LIN {X 0.155,Y -381.645,Z 884.457,A 0.000,B 0.000,C 90.000,E1 82.186} C_DIS
LIN {X -0.158,Y -370.473,Z 884.445,A 0.000,B 0.000,C 90.000,E1 80.208} C_DIS
LIN {X 0.019,Y -359.375,Z 884.434,A 0.000,B 0.000,C 90.000,E1 78.117} C_DIS
LIN {X 0.176,Y -348.139,Z 884.422,A 0.000,B 0.000,C 90.000,E1 75.992} C_DIS
LIN {X -0.033,Y -333.953,Z 884.407,A 0.000,B 0.000,C 90.000,E1 73.268} C_DIS
LIN {X 0.132,Y -321.822,Z 884.393,A 0.000,B 0.000,C 90.000,E1 70.732} C_DIS
LIN {X -0.076,Y -310.040,Z 884.379,A 0.000,B 0.000,C 90.000,E1 68.209} C_DIS
LIN {X -0.162,Y -298.515,Z 884.364,A 0.000,B 0.000,C 90.000,E1 65.613} C_DIS
LIN {X -0.024,Y -288.345,Z 884.351,A 0.000,B 0.000,C 90.000,E1 63.256} C_DIS
LIN {X -0.059,Y -279.650,Z 884.340,A 0.000,B 0.000,C 90.000,E1 61.229} C_DIS
LIN {X 0.058,Y -269.622,Z 884.327,A 0.000,B 0.000,C 90.000,E1 58.791} C_DIS
LIN {X 0.167,Y -257.412,Z 884.309,A 0.000,B 0.000,C 90.000,E1 55.595} C_DIS
LIN {X -0.046,Y -246.324,Z 884.291,A 0.000,B 0.000,C 90.000,E1 52.396} C_DIS
LIN {X -0.093,Y -236.431,Z 884.273,A 0.000,B 0.000,C 90.000,E1 49.094} C_DIS
LIN {X -0.023,Y -226.392,Z 884.252,A 0.000,B 0.000,C 90.000,E1 45.324} C_DIS
LIN {X 0.065,Y -218.832,Z 884.235,A 0.000,B 0.000,C 90.000,E1 42.243} C_DIS
LIN {X 0.001,Y -211.752,Z 884.218,A 0.000,B 0.000,C 90.000,E1 39.152} C_DIS
LIN {X -0.044,Y -205.062,Z 884.200,A 0.000,B 0.000,C 90.000,E1 36.011} C_DIS
LIN {X -0.048,Y -197.427,Z 884.178,A 0.000,B 0.000,C 90.000,E1 32.005} C_DIS
LIN {X -0.016,Y -191.938,Z 884.160,A 0.000,B 0.000,C 90.000,E1 28.743} C_DIS
LIN {X -0.059,Y -187.088,Z 884.141,A 0.000,B 0.000,C 90.000,E1 25.463} C_DIS
LIN {X 0.055,Y -182.941,Z 884.123,A 0.000,B 0.000,C 90.000,E1 22.099} C_DIS
LIN {X -0.046,Y -178.754,Z 884.099,A 0.000,B 0.000,C 90.000,E1 17.928} C_DIS
LIN {X 0.072,Y -175.685,Z 884.076,A 0.000,B 0.000,C 90.000,E1 13.647} C_DIS
LIN {X -0.042,Y -173.199,Z 884.043,A 0.000,B 0.000,C 90.000,E1 7.701} C_DIS
LIN {X -0.002,Y -174.181,Z 883.974,A 0.000,B 0.000,C 90.000,E1 355.241} C_DIS
LIN {X 0.048,Y -177.020,Z 883.945,A 0.000,B 0.000,C 90.000,E1 350.095} C_DIS
LIN {X -0.051,Y -180.525,Z 883.921,A 0.000,B 0.000,C 90.000,E1 345.880} C_DIS
LIN {X 0.013,Y -184.235,Z 883.903,A 0.000,B 0.000,C 90.000,E1 342.489} C_DIS
LIN {X -0.016,Y -188.687,Z 883.884,A 0.000,B 0.000,C 90.000,E1 339.156} C_DIS
LIN {X -0.007,Y -193.912,Z 883.866,A 0.000,B 0.000,C 90.000,E1 335.845} C_DIS
LIN {X 0.036,Y -199.724,Z 883.848,A 0.000,B 0.000,C 90.000,E1 332.564} C_DIS
LIN {X 0.062,Y -205.908,Z 883.830,A 0.000,B 0.000,C 90.000,E1 329.331} C_DIS
LIN {X -0.006,Y -212.491,Z 883.812,A 0.000,B 0.000,C 90.000,E1 326.167} C_DIS
LIN {X -0.086,Y -219.576,Z 883.795,A 0.000,B 0.000,C 90.000,E1 323.050} C_DIS
LIN {X 0.053,Y -228.296,Z 883.775,A 0.000,B 0.000,C 90.000,E1 319.542} C_DIS
LIN {X -0.053,Y -236.907,Z 883.758,A 0.000,B 0.000,C 90.000,E1 316.539} C_DIS
LIN {X 0.043,Y -247.810,Z 883.740,A 0.000,B 0.000,C 90.000,E1 313.176} C_DIS
LIN {X -0.047,Y -259.881,Z 883.722,A 0.000,B 0.000,C 90.000,E1 309.930} C_DIS
LIN {X -0.058,Y -273.148,Z 883.704,A 0.000,B 0.000,C 90.000,E1 306.744} C_DIS
LIN {X -0.004,Y -287.626,Z 883.687,A 0.000,B 0.000,C 90.000,E1 303.627} C_DIS
LIN {X 0.068,Y -303.533,Z 883.670,A 0.000,B 0.000,C 90.000,E1 300.590} C_DIS
LIN {X 0.089,Y -319.062,Z 883.656,A 0.000,B 0.000,C 90.000,E1 297.975} C_DIS
LIN {X -0.146,Y -331.909,Z 883.645,A 0.000,B 0.000,C 90.000,E1 296.104} C_DIS
LIN {X 0.198,Y -353.097,Z 883.629,A 0.000,B 0.000,C 90.000,E1 293.259} C_DIS
LIN {X -0.022,Y -378.121,Z 883.613,A 0.000,B 0.000,C 90.000,E1 290.355} C_DIS
LIN {X -0.121,Y -401.386,Z 883.599,A 0.000,B 0.000,C 90.000,E1 287.873} C_DIS
LIN {X 0.163,Y -414.282,Z 883.592,A 0.000,B 0.000,C 90.000,E1 286.496} C_DIS
LIN {X 0.162,Y -424.288,Z 883.586,A 0.000,B 0.000,C 90.000,E1 285.426} C_DIS
LIN {X -0.145,Y -436.474,Z 883.578,A 0.000,B 0.000,C 90.000,E1 284.120} C_DIS
LIN {X 0.036,Y -447.938,Z 883.571,A 0.000,B 0.000,C 90.000,E1 282.771} C_DIS
LIN {X 0.134,Y -456.587,Z 883.565,A 0.000,B 0.000,C 90.000,E1 281.715} C_DIS
LIN {X -0.123,Y -464.599,Z 883.559,A 0.000,B 0.000,C 90.000,E1 280.715} C_DIS
LIN {X 0.079,Y -471.996,Z 883.554,A 0.000,B 0.000,C 90.000,E1 279.670} C_DIS
LIN {X 0.037,Y -477.077,Z 883.550,A 0.000,B 0.000,C 90.000,E1 278.916} C_DIS
LIN {X 0.044,Y -481.563,Z 883.545,A 0.000,B 0.000,C 90.000,E1 278.163} C_DIS
LIN {X 0.084,Y -485.361,Z 883.541,A 0.000,B 0.000,C 90.000,E1 277.409} C_DIS
LIN {X -0.213,Y -487.491,Z 883.538,A 0.000,B 0.000,C 90.000,E1 276.947} C_DIS
LIN {X -0.012,Y -489.311,Z 883.536,A 0.000,B 0.000,C 90.000,E1 276.429} C_DIS
LIN {X 0.196,Y -490.727,Z 883.533,A 0.000,B 0.000,C 90.000,E1 275.910} C_DIS
LIN {X -0.121,Y -491.835,Z 883.530,A 0.000,B 0.000,C 90.000,E1 275.454} C_DIS
LIN {X 0.108,Y -492.509,Z 883.527,A 0.000,B 0.000,C 90.000,E1 274.935} C_DIS
LIN {X -0.150,Y -492.819,Z 883.525,A 0.000,B 0.000,C 90.000,E1 274.473} C_DIS
LIN {X 0.085,Y -492.708,Z 883.522,A 0.000,B 0.000,C 90.000,E1 273.955} C_DIS
LIN {X -0.203,Y -492.129,Z 883.519,A 0.000,B 0.000,C 90.000,E1 273.498} C_DIS
LIN {X 0.030,Y -491.139,Z 883.517,A 0.000,B 0.000,C 90.000,E1 272.980} C_DIS
LIN {X 0.232,Y -489.687,Z 883.514,A 0.000,B 0.000,C 90.000,E1 272.465} C_DIS
LIN {X -0.058,Y -487.663,Z 883.511,A 0.000,B 0.000,C 90.000,E1 272.007} C_DIS
LIN {X 0.148,Y -485.102,Z 883.508,A 0.000,B 0.000,C 90.000,E1 271.489} C_DIS
LIN {X -0.164,Y -481.839,Z 883.506,A 0.000,B 0.000,C 90.000,E1 271.031} C_DIS
LIN {X -0.008,Y -477.794,Z 883.503,A 0.000,B 0.000,C 90.000,E1 270.516} C_DIS
LIN {X 0.125,Y -472.798,Z 883.500,A 0.000,B 0.000,C 90.000,E1 270.000} C_DIS
LIN {X -0.082,Y -466.956,Z 883.497,A 0.000,B 0.000,C 90.000,E1 269.542} C_DIS
LIN {X 0.188,Y -460.755,Z 883.495,A 0.000,B 0.000,C 90.000,E1 269.083} C_DIS
LIN {X -0.018,Y -454.114,Z 883.493,A 0.000,B 0.000,C 90.000,E1 268.740} C_DIS
LIN {X -0.217,Y -447.146,Z 883.491,A 0.000,B 0.000,C 90.000,E1 268.453} C_DIS
LIN {X 0.008,Y -439.698,Z 883.490,A 0.000,B 0.000,C 90.000,E1 268.165} C_DIS
LIN {X 0.193,Y -431.865,Z 883.489,A 0.000,B 0.000,C 90.000,E1 267.936} C_DIS
LIN {X -0.098,Y -423.771,Z 883.488,A 0.000,B 0.000,C 90.000,E1 267.822} C_DIS
LIN {X -0.076,Y -413.438,Z 883.487,A 0.000,B 0.000,C 90.000,E1 267.707} C_DIS
LIN {X 0.205,Y -409.860,Z 883.487,A 0.000,B 0.000,C 90.000,E1 267.650} C_DIS
LIN {X 0.062,Y -181.074,Z 883.487,A 0.000,B 0.000,C 90.000,E1 267.650} C_DIS
LIN {X -0.082,Y -180.881,Z 883.473,A 0.000,B 0.000,C 90.000,E1 265.122} C_DIS
LIN {X -0.022,Y -179.000,Z 883.445,A 0.000,B 0.000,C 90.000,E1 260.038} C_DIS
LIN {X 0.072,Y -178.596,Z 883.440,A 0.000,B 0.000,C 90.000,E1 259.162} C_DIS
LIN {X -0.034,Y -175.648,Z 883.412,A 0.000,B 0.000,C 90.000,E1 254.102} C_DIS
LIN {X -0.028,Y -172.367,Z 883.388,A 0.000,B 0.000,C 90.000,E1 249.826} C_DIS
LIN {X -0.014,Y -171.158,Z 883.378,A 0.000,B 0.000,C 90.000,E1 248.103} C_DIS
LIN {X 0.029,Y -167.457,Z 883.354,A 0.000,B 0.000,C 90.000,E1 243.768} C_DIS
LIN {X -0.036,Y -166.853,Z 883.349,A 0.000,B 0.000,C 90.000,E1 242.922} C_DIS
LIN {X 0.028,Y -162.839,Z 883.325,A 0.000,B 0.000,C 90.000,E1 238.535} C_DIS
LIN {X 0.003,Y -161.522,Z 883.315,A 0.000,B 0.000,C 90.000,E1 236.786} C_DIS
LIN {X 0.043,Y -157.521,Z 883.291,A 0.000,B 0.000,C 90.000,E1 232.351} C_DIS
LIN {X -0.024,Y -155.546,Z 883.276,A 0.000,B 0.000,C 90.000,E1 229.703} C_DIS
LIN {X 0.019,Y -151.839,Z 883.251,A 0.000,B 0.000,C 90.000,E1 225.202} C_DIS
LIN {X -0.074,Y -150.057,Z 883.236,A 0.000,B 0.000,C 90.000,E1 222.528} C_DIS
LIN {X -0.040,Y -146.868,Z 883.211,A 0.000,B 0.000,C 90.000,E1 217.971} C_DIS
LIN {X -0.051,Y -145.452,Z 883.196,A 0.000,B 0.000,C 90.000,E1 215.231} C_DIS
LIN {X 0.063,Y -142.870,Z 883.170,A 0.000,B 0.000,C 90.000,E1 210.590} C_DIS
LIN {X -0.011,Y -141.487,Z 883.150,A 0.000,B 0.000,C 90.000,E1 206.924} C_DIS
LIN {X -0.026,Y -139.384,Z 883.113,A 0.000,B 0.000,C 90.000,E1 200.429} C_DIS
LIN {X -0.037,Y -138.838,Z 883.098,A 0.000,B 0.000,C 90.000,E1 197.638} C_DIS
LIN {X 0.023,Y -138.353,Z 883.056,A 0.000,B 0.000,C 90.000,E1 190.141} C_DIS
LIN {X 0.018,Y -139.522,Z 883.005,A 0.000,B 0.000,C 90.000,E1 180.802} C_DIS
LIN {X -0.041,Y -141.185,Z 882.973,A 0.000,B 0.000,C 90.000,E1 175.241} C_DIS
LIN {X 0.071,Y -142.563,Z 882.958,A 0.000,B 0.000,C 90.000,E1 172.413} C_DIS
LIN {X -0.004,Y -144.847,Z 882.932,A 0.000,B 0.000,C 90.000,E1 167.825} C_DIS
LIN {X -0.019,Y -147.471,Z 882.912,A 0.000,B 0.000,C 90.000,E1 164.157} C_DIS
LIN {X 0.009,Y -150.055,Z 882.892,A 0.000,B 0.000,C 90.000,E1 160.496} C_DIS
LIN {X 0.013,Y -153.400,Z 882.872,A 0.000,B 0.000,C 90.000,E1 156.869} C_DIS
LIN {X 0.060,Y -155.931,Z 882.857,A 0.000,B 0.000,C 90.000,E1 154.152} C_DIS
LIN {X 0.033,Y -159.798,Z 882.837,A 0.000,B 0.000,C 90.000,E1 150.589} C_DIS
LIN {X 0.019,Y -162.038,Z 882.827,A 0.000,B 0.000,C 90.000,E1 148.820} C_DIS
LIN {X -0.007,Y -166.234,Z 882.807,A 0.000,B 0.000,C 90.000,E1 145.308} C_DIS
LIN {X -0.006,Y -171.250,Z 882.788,A 0.000,B 0.000,C 90.000,E1 141.823} C_DIS
LIN {X -0.083,Y -176.139,Z 882.769,A 0.000,B 0.000,C 90.000,E1 138.405} C_DIS
LIN {X 0.034,Y -180.407,Z 882.755,A 0.000,B 0.000,C 90.000,E1 135.810} C_DIS
LIN {X 0.009,Y -185.814,Z 882.736,A 0.000,B 0.000,C 90.000,E1 132.447} C_DIS
LIN {X 0.064,Y -190.433,Z 882.722,A 0.000,B 0.000,C 90.000,E1 129.930} C_DIS
LIN {X 0.064,Y -193.263,Z 882.713,A 0.000,B 0.000,C 90.000,E1 128.257} C_DIS
LIN {X 0.062,Y -294.293,Z 882.713,A 0.000,B 0.000,C 90.000,E1 128.257} C_DIS
LIN {X 0.031,Y -296.735,Z 882.712,A 0.000,B 0.000,C 90.000,E1 128.222} C_DIS
LIN {X 0.123,Y -300.631,Z 882.711,A 0.000,B 0.000,C 90.000,E1 128.016} C_DIS
LIN {X -0.021,Y -302.926,Z 882.710,A 0.000,B 0.000,C 90.000,E1 127.855} C_DIS
LIN {X 0.169,Y -306.088,Z 882.708,A 0.000,B 0.000,C 90.000,E1 127.443} C_DIS
LIN {X -0.021,Y -308.030,Z 882.706,A 0.000,B 0.000,C 90.000,E1 127.156} C_DIS
LIN {X 0.035,Y -309.544,Z 882.705,A 0.000,B 0.000,C 90.000,E1 126.824} C_DIS
LIN {X 0.006,Y -310.752,Z 882.703,A 0.000,B 0.000,C 90.000,E1 126.503} C_DIS
LIN {X -0.035,Y -321.948,Z 882.683,A 0.000,B 0.000,C 90.000,E1 122.959} C_DIS
LIN {X -0.150,Y -332.474,Z 882.667,A 0.000,B 0.000,C 90.000,E1 120.129} C_DIS
LIN {X -0.017,Y -344.363,Z 882.652,A 0.000,B 0.000,C 90.000,E1 117.308} C_DIS
LIN {X -0.164,Y -357.712,Z 882.636,A 0.000,B 0.000,C 90.000,E1 114.591} C_DIS
LIN {X -0.166,Y -370.904,Z 882.623,A 0.000,B 0.000,C 90.000,E1 112.206} C_DIS
LIN {X -0.128,Y -385.441,Z 882.610,A 0.000,B 0.000,C 90.000,E1 109.866} C_DIS
LIN {X -0.110,Y -401.428,Z 882.598,A 0.000,B 0.000,C 90.000,E1 107.583} C_DIS
LIN {X -0.191,Y -418.977,Z 882.585,A 0.000,B 0.000,C 90.000,E1 105.371} C_DIS
LIN {X 0.072,Y -438.184,Z 882.573,A 0.000,B 0.000,C 90.000,E1 103.175} C_DIS
LIN {X -0.149,Y -458.338,Z 882.562,A 0.000,B 0.000,C 90.000,E1 101.186} C_DIS
LIN {X 0.169,Y -466.052,Z 882.558,A 0.000,B 0.000,C 90.000,E1 100.433} C_DIS
LIN {X 0.207,Y -468.379,Z 882.557,A 0.000,B 0.000,C 90.000,E1 100.197} C_DIS
LIN {X 0.244,Y -470.138,Z 882.555,A 0.000,B 0.000,C 90.000,E1 99.962} C_DIS
LIN {X 0.095,Y -471.606,Z 882.554,A 0.000,B 0.000,C 90.000,E1 99.726} C_DIS
LIN {X -0.133,Y -472.702,Z 882.553,A 0.000,B 0.000,C 90.000,E1 99.500} C_DIS
LIN {X 0.050,Y -473.998,Z 882.550,A 0.000,B 0.000,C 90.000,E1 98.973} C_DIS
LIN {X 0.164,Y -474.281,Z 882.547,A 0.000,B 0.000,C 90.000,E1 98.454} C_DIS
LIN {X -0.180,Y -473.600,Z 882.544,A 0.000,B 0.000,C 90.000,E1 97.992} C_DIS
END
